pt := ADR(oct);
stop := LEN(oct);
FOR I := 1 TO stop DO
	(* read the first character and subtract 48 to get value in decimal 0 = 48 *)
	x := pt^;
	(* calculate the value of the digit *)
	IF X > 47 AND x < 56 THEN
		OCT_TO_BYTE := SHL(OCT_TO_BYTE,3) + X - 48;
	END_IF;
	pt := pt + 1;
END_FOR;



(* revision histroy
hm	18. jun. 2008	rev 1.0
	original release

hm	20. sep. 2008	rev 1.1
	changed length of input string from 20 to 10

*)

END_FUNCTION

// POUs/String/HEX_TO_BYTE
FUNCTION HEX_TO_BYTE : BYTE
VAR_INPUT
	HEX : STRING(5);
END_VAR
VAR
	pt : POINTER TO BYTE;
	i: INT;
	X: BYTE;
	stop: INT;
END_VAR

(*
version 1.1	20. sep. 2008
programmer 	hugo
tested by		oscat

HEX_TO_BYTE converts a Hexadecimal string into a byte.

*)

pt := ADR(hex);
stop := LEN(hex);
FOR I := 1 TO stop DO
	(* read the first character and subtract 48 to get value in decimal 0 = 48 *)
	x := pt^;
	(* calculate the value of the digit *)
	IF X > 47 AND x < 58 THEN
		HEX_TO_BYTE := SHL(HEX_TO_BYTE,4) + X - 48;
	ELSIF X > 64 AND X < 71 THEN
		HEX_TO_BYTE := SHL(HEX_TO_BYTE,4) + X - 55;
	ELSIF X > 96 AND X < 103 THEN
		HEX_TO_BYTE := SHL(HEX_TO_BYTE,4) + X - 87;
	END_IF;
	pt := pt + 1;
END_FOR;




(* revision histroy
hm	18. jun. 2008	rev 1.0
	original release

hm	20. sep.2008	rev 1.1
	changed length of input string from 20 to 5

*)

END_FUNCTION

// POUs/String/FSTRING_TO_DT
FUNCTION FSTRING_TO_DT : DT
VAR_INPUT
	SDT : STRING(60);
	FMT : STRING(60);
END_VAR
VAR CONSTANT
	ignore: STRING(1) := '*';  (* ignore character is * *)
	fchar : STRING(1) := '#';  (* format character is # *)
END_VAR
VAR
	c: STRING(1);
	tmp: STRING(20);
	end: INT;
	dy : INT := 1970;
	dm : INT := 1;
	dd : INT := 1;
	th : INT;
	tm : INT;
	ts : INT;
END_VAR


(*
version 1.0	24. sep. 2008
programmer 	hugo
tested by	oscat

FSTRING_TO_DT converts Formatted String into a DT value.

*)

(* scan input string *)
WHILE fmt <> '' DO
	c := LEFT(fmt,1);
	IF c = ignore THEN
		(* skip ignore characters *)
		fmt := DELETE(fmt,1,1);
		sdt := DELETE(sdt,1,1);
	ELSIF C = fchar THEN
		(* format chracter found skip format char and read identifier *)
		(* store format identifier in c and skip to next char in fmt *)
		c := MID(fmt,1,2);
		fmt := DELETE(fmt,2,1);
		(* extract the substring until the end of sdt or to next char of fmt *)
		IF fmt = '' THEN
			tmp := sdt;
		ELSE
			(* serach for end of substring *)
			end := FIND(sdt, LEFT(fmt,1))-1;
			tmp := LEFT(sdt, end);
			sdt := DELETE(sdt, end,1);
		END_IF;
		(* extract information from substring *)
		IF c = 'Y' THEN
			dy := STRING_TO_INT(tmp);
			IF dy < 100 THEN dy := dy + 2000; END_IF;
		ELSIF c = 'M' THEN
			dm := STRING_TO_INT(tmp);
		ELSIF c = 'N' THEN
			dm := FSTRING_TO_MONTH(tmp,0);
		ELSIF c = 'D' THEN
			dd := STRING_TO_INT(tmp);
		ELSIF c = 'h' THEN
			th := STRING_TO_INT(tmp);
		ELSIF c = 'm' THEN
			tm := STRING_TO_INT(tmp);
		ELSIF c = 's' THEN
			ts := STRING_TO_INT(tmp);
		END_IF;
	ELSIF c = LEFT(sdt,1) THEN
		(* skip matching characters *)
		fmt := DELETE(fmt,1,1);
		sdt := DELETE(sdt,1,1);
	ELSE
		RETURN;
	END_IF;
END_WHILE;

FSTRING_TO_DT := SET_DT(dy,dm,dd,th,tm,ts);


(* revision histroy
hm	24. sep. 2008	rev 1.0
	original release


*)

END_FUNCTION

// POUs/String/FSTRING_TO_MONTH
FUNCTION FSTRING_TO_MONTH : INT
VAR_INPUT
	MTH : STRING(20);
	LANG : INT;
END_VAR
VAR
	lx: INT;
END_VAR


(*
version 1.2	25. oct 2008
programmer 	hugo
tested by	oscat

FSTRING_TO_MONTH converts a string into a month, the string can be a name for the month or a number.
the function is language sensitve when LANG > 1 and checks for all languages when LANG = 0

*)

IF LANG = 0 THEN lx := LANGUAGE.DEFAULT; ELSE lx := MIN(LANG, LANGUAGE.LMAX); END_IF;
MTH := TRIM(mth);
MTH := CAPITALIZE(LOWERCASE(MTH));

FOR FSTRING_TO_MONTH := 1 TO 12 DO
	IF MTH = language.MONTHS[lx, FSTRING_TO_MONTH] THEN RETURN; END_IF;
	IF MTH = language.MONTHS3[lx, FSTRING_TO_MONTH] THEN RETURN; END_IF;
END_FOR;

(* since no name matched try to decode as integer *)
FSTRING_TO_MONTH := STRING_TO_INT(MTH);




(* revision histroy
hm	25. sep. 2008	rev 1.0
	original release

hm	19. oct. 2008	rev 1.1
	changed language setup constants

hm	25. oct. 2008	rev 1.2
	optimized code
*)

END_FUNCTION

// POUs/String/FSTRING_TO_DWORD
FUNCTION FSTRING_TO_DWORD : DWORD
VAR_INPUT
	IN : STRING(40);
END_VAR


(*
version 1.1	20. sep. 2008
programmer 	hugo
tested by		oscat

FSTRING_TO_BYTE converts a formatted string into a byte.
the string can be of the form 2#01010, 8#7234, 16#2AD3 and 1234

*)

IF LEFT(IN, 2) = '2#' THEN
	(* we need to convert binary *)
	FSTRING_TO_DWORD := BIN_TO_DWORD(RIGHT(in, LEN(in) - 2));
ELSIF LEFT(in, 2) = '8#' THEN
	(* weneed to convert octals *)
	FSTRING_TO_DWORD := OCT_TO_DWORD(RIGHT(in, LEN(in) - 2));
ELSIF LEFT(in, 3) = '16#' THEN
	(* we need to convert hexadecimal *)
	FSTRING_TO_DWORD := HEX_TO_DWORD(RIGHT(in, LEN(in) - 3));
ELSE
	(* we assume decimal representation *)
	FSTRING_TO_DWORD := DEC_TO_DWORD(CLEAN(in,'0123456789'));
END_IF;


(* revision histroy
hm	18. jun. 2008	rev 1.0
	original release

hm	20. sep. 2008	rev 1.1
	changed length of input dtring from 20 to 40


*)

END_FUNCTION

// POUs/String/OCT_TO_DWORD
FUNCTION OCT_TO_DWORD : DWORD
VAR_INPUT
	OCT : STRING(20);
END_VAR
VAR
	pt : POINTER TO BYTE;
	i: INT;
	X: BYTE;
	stop: INT;
END_VAR

(*
version 1.0	18. jun 2008
programmer 	hugo
tested by	oscat

OCT_TO_DWORD converts a octagonal string into a dword.

*)

pt := ADR(oct);
stop := LEN(oct);
FOR I := 1 TO stop DO
	(* read the first character and subtract 48 to get value in decimal 0 = 48 *)
	x := pt^;
	(* calculate the value of the digit *)
	IF X > 47 AND x < 56 THEN
		OCT_TO_DWORD := SHL(OCT_TO_DWORD,3) + X - 48;
	END_IF;
	pt := pt + 1;
END_FOR;




(* revision histroy
hm	18. jun. 2008	rev 1.0
	original release


*)

END_FUNCTION

// POUs/String/HEX_TO_DWORD
FUNCTION HEX_TO_DWORD : DWORD
VAR_INPUT
	Hex : STRING(20);
END_VAR
VAR
	pt : POINTER TO BYTE;
	i: INT;
	X: BYTE;
	stop: INT;
END_VAR

(*
version 1.4	18. jun. 2008
programmer 	hugo
tested by	tobias

HEX_TO_DWORD converts a Hexadecimal string into a DWORD.

*)

pt := ADR(hex);
stop := LEN(hex);
FOR I := 1 TO stop DO
	(* read the first character and subtract 48 to get value in decimal 0 = 48 *)
	x := pt^;
	(* calculate the value of the digit *)
	IF X > 47 AND x < 58 THEN
		HEX_TO_DWORD := SHL(HEX_TO_DWORD,4) + X - 48;
	ELSIF X > 64 AND X < 71 THEN
		HEX_TO_DWORD := SHL(HEX_TO_DWORD,4) + X - 55;
	ELSIF X > 96 AND X < 103 THEN
		HEX_TO_DWORD := SHL(HEX_TO_DWORD,4) + X - 87;
	END_IF;
	pt := pt + 1;
END_FOR;



(* revision histroy
hm	2.10.2007		rev 1.0
	original release

hm	19.11.2007		rev 1.1
	changed type of function from int to dword

hm 	4. mar 2008		rev 1.2
	added support for a..f and return 0 for invalid string

hm	29. mar. 2008	rev 1.3
	changed STRING to STRING(8)

hm	18. jun. 2008	rev 1.4
	changed input hex to STRING(20)
	function now ignores wrong characters
*)

END_FUNCTION

// POUs/String/FSTRING_TO_WEEK
FUNCTION FSTRING_TO_WEEK : BYTE
VAR_INPUT
	WEEK : STRING(60);
	LANG : INT;
END_VAR
VAR
	pos: INT;
END_VAR


(*
version 1.1	25. oct. 2008
programmer 	hugo
tested by	oscat

FSTRING_TO_WEEK converts a list of weekdays into a byte where each bit represents a day of the week.
bit 6 = mo, 0 = su;

*)

pos := FIND(WEEK, ',');
WHILE pos > 0 DO
	FSTRING_TO_WEEK := FSTRING_TO_WEEK OR SHR(BYTE#128, FSTRING_TO_WEEKDAY(MID(WEEK, pos - 1, 1), LANG));
	WEEK := RIGHT(WEEK, LEN(Week) - pos);
	pos := FIND(WEEK, ',');
END_WHILE;
FSTRING_TO_WEEK := (FSTRING_TO_WEEK OR SHR(BYTE#128, FSTRING_TO_WEEKDAY(WEEK, LANG))) AND BYTE#127;


(* revision histroy
hm	18. jun. 2008	rev 1.0
	original release

hm	25. oct. 2008	rev 1.1
	using language defauls and input lang
*)

END_FUNCTION

// POUs/String/FSTRING_TO_WEEKDAY
FUNCTION FSTRING_TO_WEEKDAY : INT
VAR_INPUT
	WDAY : STRING(20);
	LANG : INT;
END_VAR
VAR
	tmp: STRING(2);
	i: INT;
	ly: INT;
END_VAR


(*
version 1.2	25. oct. 2008
programmer 	hugo
tested by	oscat

FSTRING_TO_WEEKDAY converts a weekday string into an integer 1..7.

*)

IF LANG = 0 THEN ly := LANGUAGE.DEFAULT; ELSE ly := MIN(LANG, LANGUAGE.LMAX); END_IF;
(* tmp needs to be calculated first otherwise find can return wrong values *)
tmp := TRIM(wday);
tmp := CAPITALIZE(LOWERCASE(tmp));
FOR i := 1 TO 7 DO
	IF language.WEEKDAYS2[ly, i] = tmp THEN
		FSTRING_TO_WEEKDAY := i;
		RETURN;
	END_IF;
END_FOR;
FSTRING_TO_WEEKDAY := STRING_TO_INT(WDAY);




(* revision histroy
hm	18. jun. 2008	rev 1.0
	original release

hm	18. jul. 2008	rev 1.1
	changed nested call of left(trim()) for compatibility reasons

hm	25. oct. 2008	rev 1.2
	using language constants
*)

END_FUNCTION

// POUs/Mathematical/functions/FT_AVG
FUNCTION_BLOCK FT_AVG
VAR_INPUT
	IN : REAL;
	E : BOOL := TRUE;
	N : INT := 32;
	RST : BOOL;
END_VAR
VAR_OUTPUT
	AVG : REAL;
END_VAR
VAR
	buff : DELAY;
	i: INT;
	init : BOOL;
END_VAR

(*
version 1.5	10. mar. 2009
programmer 	hugo
tested by		oscat

this function calculates the moving average over n samples from a sequential input
the input values are shifted into an N deep buffer and the avg of this buffer is diplayed at anytime on the output.
a rst will load the buffer with the current in value..

*)

(* limit n to a max of 32 because delay can do max 32 cycles *)
buff.N := LIMIT(0, N, 32);

IF NOT init OR rst THEN
	FOR i := 1 TO N DO
		buff(in := in);
	END_FOR;
	avg := in;
	init := TRUE;
ELSIF E THEN
	buff(in := in);
	avg := avg + (in - buff.out ) / INT_TO_REAL(N);
END_IF;

(* revision history

hm	7. jan. 2007	rev 1.1
	chaged rst logic to load the buffer with the actual input value instead of 0.
	added en input to allow better control of signal flow
	added init to load the buffer with in at startup to avoid rampup at beginning.
	deleted unused variable cnt.

hm	14. jun. 2008	rev 1.2
	set default for input en = TRUE and N = 32

hm	10. oct. 2008	rev 1.3
	improved performance

hm	18. oct. 2008	rev 1.4
	changed input en to e for compatibility reasons

hm	10. mar. 2009	rev 1.5
	added type conversion for compatibility reasons

*)

END_FUNCTION_BLOCK

// POUs/Engineering/control/FT_IMP
FUNCTION_BLOCK FT_IMP
VAR_INPUT
	in : REAL;
	T : TIME;
	K : REAL := 1.0;
END_VAR
VAR_OUTPUT
	out : REAL;
END_VAR
VAR
	t1 : FT_PT1;
END_VAR

(*
version 1.1	3 Jan 2007
programmer 	hugo
tested by	oscat

FT_IMP is 	an impulse filter (high pass filter) with the time T and factor K.
 
*)

T1(in:= in, T:=T);
out := (in - t1.out) * K;

(*
hm 3.1.2007	rev 1.1
	added factor K

*)

END_FUNCTION_BLOCK

// POUs/Engineering/control/FT_INT2
FUNCTION_BLOCK FT_INT2
VAR_INPUT
	IN : REAL;
	K : REAL := 1.0;
	RUN : BOOL := TRUE;
	RST : BOOL;
	OUT_MIN : REAL := -1.0E38;
	OUT_MAX : REAL := 1.0E38;
END_VAR
VAR_OUTPUT
	OUT : REAL;
	LIM : BOOL;
END_VAR
VAR
	integ: INTEGRATE;
	ix : REAL;
	val : REAL2;
END_VAR


(*
version 1.2	11. mar. 2009
programmer 	hugo
tested by		oscat

FT_int2 is an integrator with input IN and factor K.
integration is only done while run = true, if run is false integration is stopped and the out remains at the last value.
if run is left unconnected, run is considered true by the function block.
the out_min and out_max values can be set to ,imit the output value range. 
the default for K is 1.
FT_INT2 has double presision accuracy (14 digits).


*)

IF RST THEN
	val := R2_SET(0.0);
	out := 0.0;
ELSE
	integ(X := IN, E := RUN, K := K, Y := ix);
	val := R2_ADD(val, ix);
	ix := 0.0;
	OUT := val.RX;
END_IF;

(* check output for limits *)
IF out > OUT_MIN AND out < OUT_MAX THEN
	LIM := FALSE;
ELSE
	OUT := LIMIT(OUT_MIN, OUT, OUT_MAX);
	val := R2_SET(OUT);
	LIM := TRUE;
END_IF;



(*	revision history
hm	2. jun. 2008	rev 1.0
	original version

hm	5. nov. 2008	rev 1.1
	rewritten code using integrate

hm	11. mar. 2009	rev 1.2
	real constants updated to new systax using dot

*)

END_FUNCTION_BLOCK

// POUs/Mathematical/Double Precision/R2_SET
FUNCTION R2_SET : REAL2
VAR_INPUT
	X : REAL;
END_VAR


(*
version 1.1	10. mar. 2009
programmer 	hugo
tested by		tobias

R2_set sets a double precision real to a single real value.

*)

R2_SET.RX := X;
R2_SET.R1 := 0.0;


(* revision history
hm	2. jun. 2008	rev 1.0
	original version

hm	10. mar. 2009	rev 1.1
	real constants updated to new systax using dot

*)

END_FUNCTION

// POUs/Mathematical/functions/FT_MIN_MAX
FUNCTION_BLOCK FT_MIN_MAX
VAR_INPUT
	in : REAL;
	rst : BOOL;
END_VAR
VAR_OUTPUT
	mx : REAL;
	mn : REAL;
END_VAR
VAR
	init: BOOL;
END_VAR

(*
version 1.0	1 sep 2006
programmer 	hugo
tested by		tobias

this function block stores the min and max value of an input signal.
when rst is true the mn and mx outputs are set to the in value.
when a rst is never active the function autoresets to the in value at startup.
since the input might not be present at first cycle the mn and mx are set during second cycle.

*)

IF rst OR NOT init THEN
	mn := in;
	mx := in;
	init := TRUE;
ELSIF in < mn THEN mn := in;
ELSIF in > mx THEN mx := in;
END_IF;

END_FUNCTION_BLOCK

// POUs/Engineering/control/FT_PD
FUNCTION_BLOCK FT_PD
VAR_INPUT
	IN : REAL;
	KP : REAL := 1.0;
	TV : REAL := 1.0;
END_VAR
VAR_OUTPUT
	Y : REAL;
END_VAR
VAR
	diff : FT_DERIV;
END_VAR

(*
version 1.0	3. jun 2008
programmer 	hugo
tested by		tobias

FT_PD is a PD controller.
The PD controller works according to the fomula Y = KP *(IN + DERIV(e) ).

*)

(* run differentiator *)
diff(IN := IN, K := TV);

(* combine both values *)
Y := KP * (diff.out + IN);



(* revision history
hm 	3. jun. 2008 	rev 1.0
	original version


*)

END_FUNCTION_BLOCK

// POUs/Engineering/control/FT_PDT1
FUNCTION_BLOCK FT_PDT1
VAR_INPUT
	IN : REAL;
	KP : REAL := 1.0;
	TV : REAL := 1.0;
	T1 : REAL := 1.0;
END_VAR
VAR_OUTPUT
	Y : REAL;
END_VAR
VAR
	diff : FT_DERIV;
	TP : FT_PT1;
END_VAR

(*
version 1.0	3. jun 2008
programmer 	hugo
tested by		tobias

FT_PD is a PD controller.
The PD controller works according to the fomula Y = KP *(IN + DERIV(e) ).

*)

(* run differentiator *)
diff(IN := IN, K := TV);

(* Run PT1 filter *)
tp(in := diff.out, T := REAL_TO_TIME(T1));

(* combine both values *)
Y := KP * (tp.out + IN);



(* revision history
hm 	3. jun. 2008 	rev 1.0
	original version


*)

END_FUNCTION_BLOCK

// POUs/Engineering/control/FT_PID
FUNCTION_BLOCK FT_PID
VAR_INPUT
	IN : REAL;
	KP : REAL := 1.0;
	TN : REAL := 1.0;
	TV : REAL := 1.0;
	ILIM_L : REAL := -1.0E38;
	ILIM_H : REAL := 1.0E38;
	IEN : BOOL := TRUE;
	RST : BOOL;
END_VAR
VAR_OUTPUT
	Y : REAL;
	LIM : BOOL;
END_VAR
VAR
	integ : FT_INT;
	diff : FT_DERIV;
END_VAR

(*
version 2.1	11. mar. 2009
programmer 	hugo
tested by		tobias

FT_PI is a PI controller.
The PID controller works according to the fomula Y = IN *(KP+ KI * INTEG(e) ).
a rst will reset the integrator to 0
ilim_h and iLim_l set the possible output range of the internal integrator.
the output flags lim will signal that the output limits are active.

default values for KP = 1, KI = 1, ILIM_L = -1E37, iLIM_H = +1E38.
*)

(* run integrator only if TN > 0 *)
IF TN > 0.0 THEN
	integ(IN := IN, K := 1.0 / TN, RUN := IEN, RST := RST, OUT_MIN := ILIM_L, OUT_MAX := ILIM_H);
ELSE
	integ(RST := FALSE);
END_IF;

(* run differentiator *)
diff(IN := IN, K := TV);

(* combine both values *)
Y := KP * (integ.Out + diff.out + IN);

(* check if integrator has reached its limits and set overflow *)
LIM := integ.LIM;



(* revision history
hm 3. jun. 2008 	rev 2.0
	original version

hm	11. mar. 2009	rev 2.1
	real constants updated to new systax using dot

*)

END_FUNCTION_BLOCK

// POUs/Engineering/control/FT_PIDW
FUNCTION_BLOCK FT_PIDW
VAR_INPUT
	IN : REAL;
	KP : REAL := 1.0;
	TN : REAL := 1.0;
	TV : REAL := 1.0;
	LIM_L : REAL := -1.0E38;
	LIM_H : REAL := 1.0E38;
	RST : BOOL;
END_VAR
VAR_OUTPUT
	Y : REAL;
	LIM : BOOL;
END_VAR
VAR
	integ : INTEGRATE;
	diff : FT_DERIV;
	YI: REAL;
END_VAR

(*
version 1.2	11. mar. 2009
programmer 	hugo
tested by		oscat

FT_PIDW is a PID controller with dynamic wind_up reset.
The PID controller works according to the fomula Y = KP *(IN + KI * INTEG(e) + DERIV(e) ).
a rst will reset the integrator to 0
lim_h and Lim_l set the possible output range of the internal integrator.
the output flags lim will signal that the output limits are active.

default values for KP = 1, KI = 1, ILIM_L = -1E37, iLIM_H = +1E38.
*)

(* run the integrator *)
IF tn = 0.0 OR rst THEN
	integ(E := FALSE, Y := YI);
	YI := 0.0;
ELSE
	integ(X := IN, K := 1.0 / TN, E := NOT LIM, Y := YI);
END_IF;

(* add up integrator and linear part *)
Y := KP * (IN + YI);

(* run differentiator *)
diff(IN := IN, K := TV);

(* set lim before differentiator is added to stop integrator if necessary *)
IF Y > LIM_L AND Y < LIM_H THEN
	LIM := FALSE;
ELSE
	LIM := TRUE;
END_IF;

(* add differential part and limit output Y *)

Y := LIMIT(LIM_L, Y + KP * diff.out, LIM_H);




(* revision history
hm 3. jun. 2008 	rev 1.0
	original version

hm	5. nov. 2008	rev 1.1
	changed code to use integrate

hm	11. mar. 2009	rev 1.2
	real constants updated to new systax using dot

*)

END_FUNCTION_BLOCK

// POUs/Engineering/control/FT_PIW
FUNCTION_BLOCK FT_PIW
VAR_INPUT
	IN : REAL;
	KP : REAL := 1.0;
	KI : REAL := 1.0;
	LIM_L : REAL := -1E38;
	LIM_H : REAL := 1E38;
	RST : BOOL;
END_VAR
VAR_OUTPUT
	Y : REAL;
	LIM : BOOL;
END_VAR
VAR
	integ : FT_INT;
END_VAR

(*
version 1.0	3. jun 2008
programmer 	hugo
tested by		tobias

FT_PIW is a PI controller.
The PID controller works according to the fomula Y = IN *(KP+ KI * INTEG(e) ).
a rst will reset the integrator to 0
ilim_h and iLim_l set the possible output range of the internal integrator.
the output flag lim will signal that the output limits are active.
the controller is equipped with anti wind_up circuitry that stops the integrator when lim_h or lim_l is reached


default values for KP = 1, KI = 1, ILIM_L = -1E37, iLIM_H = +1E38.
*)

(* run integrator *)
integ(IN := IN, K := KI, RUN := NOT LIM, RST := RST);

(* set output value *)
Y := KP * IN + integ.Out;

(* check for limits and set integrator for anti wind up *)
IF Y < LIM_L THEN
	Y := LIM_L;
	LIM := TRUE;
ELSIF Y > LIM_H THEN
	Y := LIM_H;
	LIM := TRUE;
ELSE
	LIM := FALSE;
END_IF;



(* revision history
hm 	3. jun. 2008 	rev 1.0
	original version


*)

END_FUNCTION_BLOCK

// POUs/Engineering/automation/FT_Profile
FUNCTION_BLOCK FT_Profile
VAR_INPUT
	K : REAL := 1.0;
	O : REAL;
	M : REAL := 1.0;
	E : BOOL;
END_VAR
VAR_INPUT CONSTANT
	value_0 : REAL;
	time_1 : TIME;
	value_1 : REAL;
	time_2 : TIME;
	value_2 : REAL;
	time_3 : TIME;
	value_3 : REAL;
	time_10 : TIME;
	value_10 : REAL;
	time_11 : TIME;
	value_11 : REAL;
	time_12 : TIME;
	value_12 : REAL;
	time_13 : TIME;
	value_13 : REAL;
END_VAR
VAR_OUTPUT
	Y : REAL;
	RUN : BOOL;
	ET : TIME;
END_VAR
VAR
	tx : TIME;
	edge : BOOL;
	state: BYTE;
	ta: TIME;
	tb: TIME;
	t0 : TIME;
	temp: REAL;
	va: REAL;
	vb: REAL;
END_VAR

(*
version 1.1	15 sep 2007
programmer 	tobias
tested by		hugo

FT_Profile generates an output signal which is defined by values over a time scale.
the different values are connected by ramps between the individual values.
a rising edge on E starts the output signal generation and E = True can delay time_3 / value_3 as long as it stays true.
an additional multiplier K can be used to multiply the output and an offset O can be added to the output dynamically.
*)

(* read system time *)
tx := DWORD_TO_TIME(T_PLC_MS());

(* determine start condition *)
IF E AND NOT edge THEN
	RUN := TRUE;
	ET := t#0s;
	t0 := tx;
	ta := tx;
	tb := multime(time_1, M);
	va := value_0;
	vb := value_1;
	temp := value_0;
	state := 1;
END_IF;
edge := E;

(* generate startup profile *)
IF run THEN
	CASE state OF
		1:	IF tx - ta >= tb THEN
				ta := ta + tb;
				tb := multime(time_2 - time_1, M);
				va := value_1;
				vb := value_2;
				temp := value_1;
				state := 2;
			ELSE
				temp := ((vb - va) * TIME_TO_REAL(tx - ta) / TIME_TO_REAL(tb) + va);
			END_IF;
		2:	IF tx - ta >= tb THEN
				ta := ta + tb;
				tb := multime(time_3 - time_2, M);
				va := value_2;
				vb := value_3;
				temp := value_2;
				state := 3;
			ELSE
				temp := ((vb - va) * TIME_TO_REAL(tx - ta) / TIME_TO_REAL(tb) + va);
			END_IF;
		3:	IF tx - ta >= tb THEN
				ta := ta + tb;
				tb := multime(time_10 - time_3, M);
				va := value_3;
				vb := value_10;
				temp := value_3;
				state := 4;
			ELSE
				temp := ((vb - va) * TIME_TO_REAL(tx - ta) / TIME_TO_REAL(tb) + va);
			END_IF;
		4 :	IF tx - ta >= tb THEN
				ta := ta + tb;
				tb := multime(time_11 - time_10, M);
				va := value_10;
				vb := value_11;
				temp := value_10;
				IF E THEN state := 5; ELSE state := 6; END_IF;
			ELSE
				temp := ((vb - va) * TIME_TO_REAL(tx - ta) / TIME_TO_REAL(tb) + va);
			END_IF;
		5:	(* extend the signal while E is true *)
			IF E THEN
				ta := tx;
			ELSE
				state := 6;
			END_IF;
		6:	IF tx - ta >= tb THEN
				ta := ta + tb;
				tb := multime(time_12 - time_11, M);
				va := value_11;
				vb := value_12;
				temp := value_11;
				state := 7;
			ELSE
				temp := ((vb - va) * TIME_TO_REAL(tx - ta) / TIME_TO_REAL(tb) + va);
			END_IF;
		7:	IF tx - ta >= tb THEN
				ta := ta + tb;
				tb := multime(time_13 - time_12, M);
				va := value_12;
				vb := value_13;
				temp := value_12;
				state := 8;
			ELSE
				temp := ((vb - va) * TIME_TO_REAL(tx - ta) / TIME_TO_REAL(tb) + va);
			END_IF;
		8:	IF tx - ta >= tb THEN
				temp := value_13;
				run := FALSE;
			ELSE
				temp := ((vb - va) * TIME_TO_REAL(tx - ta) / TIME_TO_REAL(tb) + va);
			END_IF;
	END_CASE;
	Y := temp * K + O;
	ET := tx - t0;
END_IF;

(* revision history
hm	27 feb 2007		rev 1.0
	original version

hm	15. sep2007		rev 1.1
	replaced Time() with T_PLC_MS for compatibility and performance reasons

*)

END_FUNCTION_BLOCK

// POUs/Engineering/control/FT_PT2
FUNCTION_BLOCK FT_PT2
VAR_INPUT
	in : REAL;
	T : TIME;
	D : REAL;
	K : REAL := 1.0;
END_VAR
VAR_OUTPUT
	out : REAL;
END_VAR
VAR
	init: BOOL;
	int1 : INTEGRATE;
	int2 : INTEGRATE;
	tn: REAL;
	I1, I2 : REAL;
	tn2: REAL;
END_VAR

(*
version 1.5	11. mar. 2009
programmer 	hugo
tested by		oscat

FT_PT2 is a 2nd grade filter with programmable times T, D and faktor K.
 
*)

(* startup initialisation *)
IF NOT init OR T = T#0s THEN
	init := TRUE;
	out := K * in;
	I2 := out;
ELSE
	TN := TIME_TO_REAL(T) * 1.0E-3;
	tn2 := TN * TN;
	int1(X := in * K / tn2 - I1 * 0.5 * D / TN - I2 / TN2, Y := I1);
	int2(X := I1,Y := I2);
	out := I2;
END_IF;


(* revision history

15.1.2007 hm		rev 1.1
	changed formula to new more acurate formula

hm 15.9.2007		rev 1.2
	deleted unused code for init system time reading tx	

hm	30.11.2007	rev 1.3
	changed out to be K * in during initialization
	avoind divide by 0 if tn = 0

hm	3. nov. 2008	rev 1.4
	optimized code and fixed a problem with init

hm	11. mar. 2009	rev 1.5
	real constants updated to new systax using dot

*)

END_FUNCTION_BLOCK

// POUs/Engineering/control/FT_TN16
FUNCTION_BLOCK FT_TN16
VAR_INPUT
	in : REAL;
	T : TIME;
END_VAR
VAR_OUTPUT
	out : REAL;
	trig : BOOL;
END_VAR
VAR
	length : INT := 16;
	X : ARRAY[0..15] OF REAL;
	cnt : INT;
	last : TIME;
	tx: TIME;
	init: BOOL;
END_VAR

(*
version 1.1	16 sep 2007
programmer 	hugo
tested by		tobias

FT_TN16 is delay function, it will delay a signal by a specified time : T and will store 16 values of in before they are put thru to out.
for higher or lower resolution please use FT_TN8 or FT_TN64 instead.
 
*)

(* read system time *)
tx := DWORD_TO_TIME(T_PLC_MS());

trig := FALSE;
IF NOT init THEN
	x[cnt] := in;
	init := TRUE;
	last := tx;
ELSIF tx - last >= T / length THEN
	IF cnt = length - 1 THEN cnt := 0; ELSE cnt := cnt + 1; END_IF;
	Out := X[cnt];
	x[cnt] := in;
	last := tx;
	Trig := TRUE;
END_IF;

(* revision history
hm		1. jan 2007	rev 1.0
	original version

hm		16. sep 2007	rev 1.1
	changes time() to T_plc_ms() for compatibility reasons

*)

END_FUNCTION_BLOCK

// POUs/Engineering/control/FT_TN8
FUNCTION_BLOCK FT_TN8
VAR_INPUT
	in : REAL;
	T : TIME;
END_VAR
VAR_OUTPUT
	out : REAL;
	trig: BOOL;
END_VAR
VAR
	length : INT := 8;
	X : ARRAY[0..7] OF REAL;
	cnt : INT;
	last : TIME;
	tx: TIME;
	init: BOOL;
END_VAR

(*
version 1.1	15 Sep 2007
programmer 	hugo
tested by		tobias

FT_TN8 is delay function, it will delay a signal by a specified time : T and will store 8 values of in before they are put thru to out.
if higher resolution is needed, pls use FT_TN16 or FT_TN64 instead.
 
*)

tx := DWORD_TO_TIME(T_PLC_MS());
trig := FALSE;
IF NOT init THEN
	x[cnt] := in;
	init := TRUE;
	last := tx;
ELSIF tx - last >= T / length THEN
	IF cnt = length - 1 THEN cnt := 0; ELSE cnt := cnt + 1; END_IF;
	Out := X[cnt];
	x[cnt] := in;
	last := tx;
	trig := TRUE;
END_IF;

(* revision history
hm		1. jan 2007		rev 1.0
	original version

hm		16. sep 2007	rev 1.1
	changes time() to T_plc_ms() for compatibility reasons

*)

END_FUNCTION_BLOCK

// POUs/Engineering/control/FT_TN64
FUNCTION_BLOCK FT_TN64
VAR_INPUT
	in : REAL;
	T : TIME;
END_VAR
VAR_OUTPUT
	out : REAL;
	trig: BOOL;
END_VAR
VAR
	length : INT := 64;
	X : ARRAY[0..63] OF REAL;
	cnt : INT;
	last : TIME;
	tx: TIME;
	init: BOOL;
END_VAR

(*
version 1.1	15 sep 2007
programmer 	hugo
tested by		tobias

FT_TN7 is delay function, it will delay a signal by a specified time : T and will store 64 values of in before they are put thru to out.
if lower resolution is needed, pls use FT_TN8 or FT_TN16 instead.
 
*)

(* read system time *)
tx := DWORD_TO_TIME(T_PLC_MS());

trig := FALSE;
IF NOT init THEN
	x[cnt] := in;
	init := TRUE;
	last := tx;
ELSIF tx - last >= T / length THEN
	IF cnt = length - 1 THEN cnt := 0; ELSE cnt := cnt + 1; END_IF;
	Out := X[cnt];
	x[cnt] := in;
	last := tx;
	trig := TRUE;
END_IF;

(* revision history
hm		1. jan 2007		rev 1.0
	original version

hm		16. sep 2007	rev 1.1
	changes time() to T_plc_ms() for compatibility reasons

*)

END_FUNCTION_BLOCK

// POUs/Mathematical/GAUSS
FUNCTION GAUSS : REAL
VAR_INPUT
	X : REAL;
	U : REAL;
	SI: REAL;
END_VAR
VAR
	temp: REAL;
	si_inv: REAL;
END_VAR


(*
version 1.2	10. mar. 2009
programmer 	hugo
tested by		tobias

this function calculates the gaussian density function

*)

temp := X - U;
si_inv := 1.0  / si;
GAUSS := EXP(Temp * Temp * si_inv * SI_inv * - 0.5) * 0.39894228 * si_inv;



(* revision hisdtory
hm	6. apr. 2008	rev 1.0
	original version

hm	27. oct. 2008	rev 1.1
	optimized performance	

hm	10. mar. 2009	rev 1.2
	real constants updated to new systax using dot

*)

END_FUNCTION

// POUs/Mathematical/GAUSSCD
FUNCTION GAUSSCD : REAL
VAR_INPUT
	X : REAL;
	U : REAL;
	SI: REAL;
END_VAR


(*
version 1.1	10. mar. 2009
programmer 	hugo
tested by		tobias

this function calculates the gaussian cumulative distribution function

*)

GAUSSCD := (ERF((X - U) / (SI * 1.414213562)) + 1.0) * 0.5;



(* revision hisdtory
hm	6. apr. 2008	rev 1.0
	original version

hm	10. mar. 2009	rev 1.1
	real constants updated to new systax using dot

*)

END_FUNCTION

// POUs/Mathematical/GDF
FUNCTION GDF : REAL
VAR_INPUT
	X : REAL;
END_VAR


(*
version 1.2	10. mar. 2009
programmer 	hugo
tested by		tobias

this function calculates the Gudermannian function.

*)

IF X = 0.0 THEN
	GDF := 0.0;
ELSIF X > 15.0 THEN
	GDF := math.PI05;
ELSIF X < -15.0 THEN
	GDF := -math.PI05;
ELSE
	GDF := ATAN(EXP(X)) * 2.0 - math.PI05;
END_IF;

(* revision history
hm	27. apr. 2008	rev 1.0
	original version

hm	18. oct. 2008	rev 1.1
	using math constants

hm	10. mar. 2009	rev 1.2
	real constants updated to new systax using dot

*)

END_FUNCTION

// POUs/Logic/generators/GEN_BIT
FUNCTION_BLOCK GEN_BIT
VAR_INPUT
	in0 : DWORD;
	in1 : DWORD;
	in2 : DWORD;
	in3 : DWORD;
	clk : BOOL;
	steps : INT;
	rep : INT;
	rst : BOOL;
END_VAR
VAR_OUTPUT
	Q0 :BOOL;
	Q1 :BOOL;
	Q2 :BOOL;
	Q3 :BOOL;
	cnt : INT;
	run : BOOL;
END_VAR
VAR
	r0: DWORD;
	r1: DWORD;
	r2: DWORD;
	r3: DWORD;
	rx : INT := 1;
END_VAR

(*
version 1.2	14. mar. 2009
programmer 	hugo
tested by		tobias

gen_bit is 4 bit sequencial pattern generator with 4 DWORD inputs and 4 serial outputs.
with the first clock pulse after a reset or after power on, bit 0 of the input DWORDS IN is present on the Outputs Q and the next clock cycle shifts to Bit 1 and so on.
the input steps defines how many bits of the input dwords will be shifted to the outputs. the sequence can be repetive when rep = 0 or any amount of repetitions can be defined with input rep.

*)

(* check if number of runs is finished or rep = 0 which means continuous *)

IF clk AND NOT rst THEN
	run := (rep = 0) OR (rx <= rep);
	IF run THEN
		(* check for step counter reached and reset to 0 if cnt = steps *)
		IF cnt = steps THEN
			cnt := 0;
		END_IF;

		(* when cnt = 0 then reload the inputs into the registers *)
		IF cnt = 0 THEN
			r0 := in0;
			r1 := in1;
			r2 := in2;
			r3 := in3;
		END_IF;

		(* when cnt < steps, shift the lowest bits to the outputs *)
		IF (cnt < steps) THEN
			Q0 := r0.0;
			Q1 := r1.0;
			Q2 := r2.0;
			Q3 := r3.0;
			r0 := SHR(r0,1);
			r1 := SHR(r1,1);
			r2 := SHR(r2,1);
			r3 := SHR(r3,1);
		END_IF;

		(* increment the step counter *)
		cnt := cnt +1;
		IF (cnt = steps) AND (rep <> 0) THEN rx := rx +1; END_IF;
		IF (rx > rep) AND (rep <> 0) THEN run := FALSE; END_IF;
	END_IF;
ELSE
	IF rst THEN
		run := FALSE;
		Q0 := FALSE;
		Q1 := FALSE;
		Q2 := FALSE;
		Q3 := FALSE;
		r0 := 0;
		r1 := 0;
		r2 := 0;
		r3 := 0;
		cnt := 0;
		rx := 1;
	END_IF;
END_IF;



(* revision histroy
hm	4 aug 2006	rev 1.0
	original version

hm 15. oct. 2008	rev 1.1
	improved performance

hm	14. mar. 2009	rev 1.2
	removed double assignments

*)

END_FUNCTION_BLOCK

// POUs/Engineering/signal generators/GEN_PW2
FUNCTION_BLOCK GEN_PW2
VAR_INPUT
	ENQ : BOOL;
	TH1 : TIME;
	TL1 : TIME;
	TH2 : TIME;
	TL2 : TIME;
	TS : BOOL;
END_VAR
VAR_OUTPUT
	Q : BOOL;
	TH : TIME;
	TL : TIME;
END_VAR
VAR
	t_high : TIME;
	t_low : TIME;
	tx : TIME;
	start : TIME;
	init : BOOL;
	et : TIME;
END_VAR

(*
version 1.1	14. mar. 2009
programmer 	hugo
tested by		oscat

GEN_PW2 generates a time TH? followed by a time TL?.
the input ts selects between 2 sets of timings for the operation.


*)

(* read system timer *)
tx := DWORD_TO_TIME(T_PLC_MS());

(* startup initialization *)
IF NOT init THEN
	start := tx;
	init := TRUE;
	TH := T#0s;
	TL := T#0s;
END_IF;

(* timing selection *)
IF TS THEN
	t_high := TH2;
	t_low := TL2;
ELSE
	t_high := TH1;
	t_low := TL1;
END_IF;

(* normal operation *)
IF ENQ THEN
	et := tx - start;
	IF NOT Q THEN
		IF et >= t_low THEN
			Q := TRUE;
			start := tx;
			TL := T#0s;
		ELSE
			TL := et;
		END_IF;
	ELSE
		IF et >= t_high THEN
			Q := FALSE;
			start := tx;
			TH := T#0s;
		ELSE
			TH := et;
		END_IF;
	END_IF;
ELSE
	Q := FALSE;
	TH := T#0s;
	TL := T#0s;
	start := tx;
END_IF;



(* revision history
hm	26. sep. 2008	rev 1.0
	original version

hm	14. mar. 2009	rev 1.1
	removed double assignments

*)

END_FUNCTION_BLOCK

// POUs/Engineering/signal generators/GEN_RDM
FUNCTION_BLOCK GEN_RDM
VAR_INPUT
	PT : TIME;
	AM : REAL := 1;
	OS : REAL;
END_VAR
VAR_OUTPUT
	Q : BOOL;
	Out : REAL;
END_VAR
VAR
	tx : TIME;
	last : TIME;
	init : BOOL;
END_VAR

(*
	version 1.1	16 sep 2007
	programmer 	oscat
	tested BY		oscat

this signal generator generates a random output. The signal is defined by period time (PT), 
amplitude (AM), offset (OS).
The Output waveform will have its max peak at AM/2 + OS and its minimum peak at -AM/2 + OS. 
The period time PT defines how often the output signal will jump to a new randow value.
The Output Q will be true for one cycle anytime the output OUT has changed

*)

(* read system time and prepare input data *)
tx := DWORD_TO_TIME(T_PLC_MS()) - last;

(* init section *)
IF NOT init THEN
	init := TRUE;
	last := tx;
	tx := t#0s;
END_IF;

(* add last if one cycle is finished *)
IF tx >= pt THEN
	last := last + pt;
	tx := tx - pt;

	(* generate output signal *)
	out := am * (RDM(0) - 0.5) + os;
	q := TRUE;
ELSE
	q := FALSE;
END_IF;

(* revision history

hm	7.2.2007		rev 1.0
	original version

hm	16.9.2007		rev 1.1
	changes time() to T_plc_ms() for compatibility reasons

*)

END_FUNCTION_BLOCK

// POUs/Engineering/signal generators/GEN_RDT
FUNCTION_BLOCK GEN_RDT

VAR_INPUT
	Enable		 : BOOL := TRUE ;
	Min_Time_ms	: TIME := t#1s ; (* min Taktzeit *)
	Max_Time_ms	: TIME := t#1.2s ; (* Max Taktzeit *)
	TP_Q		 : TIME := t#100ms ; (* Zeit Ausgang auf TRUE *)
END_VAR
VAR_OUTPUT
	xQ		 : BOOL ;
END_VAR
VAR
	(* Taktgenerator Simulation *)
	tonRDMTimer	: TON ; (* Zeitbaustein Taktgenerator *)
	tof_xQ		: TOF ; (* Ausschaltverzögerung Taktgenerator *)
	tRDMTime	: TIME ; (* Sollzeit *)
	rRDMTime	: REAL ; (* Zufalswert Timer *)
END_VAR

(*
version 1.1	16 mar. 2008
programmer 	J. Schohaus
tested by		Hugo

RDMT generates a defined pulse with pulse width TP_Q at random times. the random time will be defined with an minimum and maximum time.

*)


(*
FUNCTION_BLOCK RDMTimer
###############################################################################
		 Ersteller / author :		 		 		 		 		 J.Schohaus
		 Datum / date:		 		 		 		 		 		 13.07.2007
###############################################################################
		 Änderungen / Datum / Ersteller :		 		 		 		 		 		 		 		 		 		 		 		 		 		 		 
		 moditication / date / author :		 		 
###############################################################################
		 Verwendete Bibliotheken		 ( * werden im Baustein nicht benötigt )
		 		 		 		 Oscat.lib
###############################################################################
Beschreibung:
*)

tonRDMTimer ( IN:= Enable , PT:= tRDMTime );
tof_xQ ( IN:= tonRDMTimer.Q , PT:= TP_Q );
XQ := tof_xq.Q;
IF tonRDMTimer.Q THEN
		 xQ := TRUE ;
		 rRDMTime := RDM ( last:= rRDMTime ) ;
		 tRDMTime := REAL_TO_TIME ( rRDMTime * DINT_TO_REAL(TIME_TO_DINT( Max_Time_ms - Min_Time_ms ) + TIME_TO_DINT(Min_Time_ms ))) ;
		 tonRDMTimer ( IN:= FALSE );
END_IF;

(* revision history
J. Schohaus	19. nov 2007	rev 1.0
	origial version

hm	16. mar. 2008			rev 1.1
	added type conversion to avoid warnings under codesys 3.0
*)

END_FUNCTION_BLOCK

// POUs/Engineering/signal generators/GEN_RMP
FUNCTION_BLOCK GEN_RMP
VAR_INPUT
	PT : TIME := t#1s;
	AM : REAL := 1.0;
	OS : REAL;
	DL : REAL;
END_VAR
VAR_OUTPUT
	Q : BOOL;
	OUT : REAL;
END_VAR
VAR
	tx : TIME;
	last : TIME;
	init : BOOL;
	temp : REAL;
	ltemp: REAL;
END_VAR

(*
	version 1.4	10. mar. 2009
	programmer 	oscat
	tested BY		oscat

this signal generator generates a ramp wave output. The ramp wave signal is defined by period time (PT), 
amplitude (AM), offset (OS) and a specific delay for the output signal (DL).
The Output waveform will have its minimum peak at OS and its maximum peak at AM + OS. 
The delay input can delay a signal up to PT, this can be useful to synchronize different generators 
and generate interleaving signals.
in addition to the analog output Out there is a second boolean output Q with is true for one cycle when the ramp starts.
*)

(* read system time and prepare input data *)
tx := DWORD_TO_TIME(T_PLC_MS()) - last;
DL := MODR(dl,1.0);
IF dl < 0.0 THEN dl := 1.0 - dl; END_IF;

(* init section *)
IF NOT init THEN
	init := TRUE;
	last := tx;
	tx := t#0s;
END_IF;

(* add last if one cycle is finished *)
IF tx >= pt THEN
	last := last + pt;
	tx := tx - pt;
END_IF;

(* generate sine wave *)
ltemp := temp;
IF pt > t#0s THEN temp := FRACT(TIME_TO_REAL(tx + MULTIME(pt, dl)) / TIME_TO_REAL(pt)); END_IF;
out := am * temp + os;

(* boolean output Q *)
Q := temp < ltemp;

(* revision history
hm	3. mar 2007		rev 1.0
	original version

hm	17 sep 2007		rev 1.1
	replaced time() with t_plc_ms for compatibilitx reasons

hm	27. nov 2007	rev 1.2
	avoid divide by 0 when pt = 0

ks	26. oct. 2008	rev 1.3
	code optimization

hm	10. mar. 2009	rev 1.4
	changed real constants to use dot syntax
*)

END_FUNCTION_BLOCK

// POUs/Engineering/signal generators/GEN_SIN
FUNCTION_BLOCK GEN_SIN
VAR_INPUT
	PT : TIME;
	AM : REAL := 1.0;
	OS : REAL;
	DL : REAL;
END_VAR
VAR_OUTPUT
	Q : BOOL;
	Out : REAL;
END_VAR
VAR
	tx : TIME;
	last : TIME;
	init : BOOL;
	temp : REAL;
END_VAR

(*
version 1.6	11. mar. 2009
programmer 	oscat
tested BY	oscat

this signal generator generates a sine wave output. The sine wave signal is defined by period time (PT), 
amplitude (AM), offset (OS) and a specific delay for the output signal (DL).
The Output waveform will have its max peak at AM/2 + OS and its minimum peak at -AM/2 + OS. 
The delay input can delay a signal up to PT, this can be useful to synchronize different generators 
and generate interleaving signals. A Cos wave can be generated accordingly.
in addition to a analog output Out there is a second boolean output Q with the corresponding binary signal.
*)

(* read system time and prepare input data *)
tx := DWORD_TO_TIME(T_PLC_MS()) - last;
DL := MODR(dl,1.0);
IF dl < 0.0 THEN dl := 1.0 - dl; END_IF;

(* init section *)
IF NOT init THEN
	init := TRUE;
	last := tx;
	tx := t#0s;
END_IF;

(* add last if one cycle is finished *)
IF tx >= pt THEN
	last := last + pt;
	tx := tx - pt;
END_IF;

(* generate sine wave *)
IF pt > t#0s THEN temp := SIN(math.PI2 * DWORD_TO_REAL(TIME_TO_DWORD(tx + MULTIME(pt, dl))) / DWORD_TO_REAL(TIME_TO_DWORD(pt))); END_IF;
out := am * 0.5 *  temp + os;

(* boolean output Q *)
q := NOT SIGN_R(temp);

(* revision history
hm	22. jan 2007	rev 1.0
	original version

hm	17 sep 2007	rev 1.1
	replaced time() with t_plc_ms for compatibilitx reasons

hm	27. nov 2007	rev 1.2
	avoid divide by 0 when pt = 0

hm	6. jan 2008		rev 1.3
	improved performance

hm	16. mar. 2008	rev 1.4
	added type conversion to avoid warnings under codesys 3.0

hm	18. oct. 2008	rev 1.5
	using math constants

hm	11. mar. 2009	rev 1.6
	changed real constants to use dot syntax

*)

END_FUNCTION_BLOCK

// POUs/Logic/generators/GEN_SQ
FUNCTION_BLOCK GEN_SQ
VAR_INPUT
	PT : TIME;
END_VAR
VAR_OUTPUT
	Q : BOOL;
END_VAR
VAR
	tn: TIME;
	tx: TIME;
	init : BOOL;
END_VAR

(*
version 1.2	18. jul. 2009
programmer 	hugo
tested by		tobias

gen_sq generates square wave signal with programmable period time.

*)

(* read system time *)
tx := DWORD_TO_TIME(T_PLC_MS());

IF tx >= tn THEN
	Q := NOT Q;
	IF init THEN
		tn := tn + DWORD_TO_TIME(SHR(TIME_TO_DWORD(PT),1));
	ELSE
		tn := tx;
		init := TRUE;
	END_IF;
END_IF;

(* revision history
hm	4. aug 2006	rev 1.0
	original version

hm	17. sep 2007	rev 1.1
	replaced time() with T_PLC_MS() for compatibility reasons

hm	18. jul. 2009	rev 1.2
	improved accuracy

*)

END_FUNCTION_BLOCK

// POUs/Engineering/signal generators/GEN_SQR
FUNCTION_BLOCK GEN_SQR
VAR_INPUT
	PT : TIME;
	AM : REAL := 1.0;
	OS : REAL;
	DC : REAL := 0.5;
	DL : REAL;
END_VAR
VAR_OUTPUT
	Q : BOOL;
	Out : REAL;
END_VAR
VAR
	tx : TIME;
	last : TIME;
	init: BOOL;
END_VAR

(*
version 1.4	11. mar. 2009
programmer 	oscat
tested BY		oscat

this signal generator generates a square wave output. The square wave signal is defined by period time (PT), 
amplitude (AM), offset (OS), duty cycle (DC) and a specific delay for the output signal (DL).
The Output waveform will switch between AM/2 + OS and -AM/2 + OS. The DC input specifies ther duty cycle, 
DC = 0 means output is low at all times and 1 means output is high at all times.
The delay input can delay a signal up to PT, this can be useful to synchronize different generators and generate interleaving signals.
in addition to a analog output Out there is a second boolean output Q.
*)

(* check dc = 1 or 0 *)
IF dc = 0.0 THEN
	out := -am * 0.5 + os;
	Q := FALSE;
	RETURN;
ELSIF dc = 1.0 THEN
	out := am * 0.5 + os;
	Q := TRUE;
	RETURN;
END_IF;

(* read system time and prepare input data *)
tx := DWORD_TO_TIME(T_PLC_MS()) - last;
DL := MODR(dl,1.0);
IF dl < 0.0 THEN dl := 1.0 - dl; END_IF;
dc := MODR(dc,1.0);
IF dc < 0.0 THEN dc := 1.0 - dc; END_IF;

(* init section *)
IF NOT init THEN
	init := TRUE;
	last := tx;
	tx := t#0s;
END_IF;

(* add last if one cycle is finished *)
IF tx >= pt THEN
	last := last + pt;
	tx := tx - pt;
END_IF;

(* check if falling or rising edge first *)
IF MULTIME(pt, dl + dc) >= pt THEN
	(* generate falling edge *)
	IF tx >= MULTIME(pt, dl + dc - 1) THEN
		out := -am * 0.5 + os;
		Q := FALSE;
	END_IF;
	(* generate rising edge *)
	IF tx >= MULTIME(pt, dl) THEN
		out := am * 0.5 + os;
		Q := TRUE;
	END_IF;
ELSE
	(* generate rising edge first *)
	IF tx >= MULTIME(pt, dl) THEN
		out := am * 0.5 + os;
		Q := TRUE;
	END_IF;
	(* generate falling edge *)
	IF tx >= MULTIME(pt, dl + dc) THEN
		out := -am * 0.5 +os;
		Q := FALSE;
	END_IF;
END_IF;

(* revision history

hm	12. feb 2007	rev 1.1
	added default value for dc = 0.5

hm	17 sep 2007	rev 1.2
	replaced time() with t_plc_ms for compatibilitx reasons

hm	6. jan 2008	rev 1.3
	improved performance

hm	11. mar. 2009	rev 1.4
	changed real constants to use dot syntax
	set default amplitude to 1.0

*)

END_FUNCTION_BLOCK

// POUs/Engineering/conversion/GEO_TO_DEG
FUNCTION GEO_TO_DEG : REAL
VAR_INPUT
	D : INT;
	M : INT;
	SEC : REAL;
END_VAR


(*
version 1.0	22. jan. 2009
programmer 	hugo
tested by		oscat

this function converts degrees, minutes seconds to decimal degrees.

*)

GEO_TO_DEG := INT_TO_REAL(D) + INT_TO_REAL(M) * 0.016666666666667 + sec * 0.00027777777777778;


(* revision histroy
hm	22. jan. 2009	rev 1.0
	original release


*)

END_FUNCTION

// POUs/Mathematical/GOLD
FUNCTION GOLD : REAL
VAR_INPUT
	X : REAL;
END_VAR


(*
version 1.1	10. mar. 2009
programmer 	hugo
tested by		tobias

this function calculates the golden function.

*)

GOLD := (X + SQRT(X*X + 4.0)) * 0.5;


(* revision history
hm	27. apr. 2008	rev 1.0
	original version

hm	10. mar. 2009	rev 1.1
	real constants updated to new systax using dot

*)

END_FUNCTION

// POUs/Logic/gate logic/GRAY_TO_BYTE
FUNCTION GRAY_TO_BYTE : BYTE
VAR_INPUT
	IN : BYTE;
END_VAR


(*
version 1.0	9. nov. 2009
programmer 	hugo
tested by		oscat

this function converts a gray code into binary

*)

GRAY_TO_BYTE := SHR(IN,4) XOR IN;
GRAY_TO_BYTE := SHR(GRAY_TO_BYTE,2) XOR GRAY_TO_BYTE;
GRAY_TO_BYTE := SHR(GRAY_TO_BYTE,1) XOR GRAY_TO_BYTE;

(* revision history
hm	9. nov. 2009	rev 1.0
	original version

*)

END_FUNCTION

// POUs/Building/HLK/HEAT_INDEX
FUNCTION HEAT_INDEX : REAL
VAR_INPUT
	T : REAL;
	RH : REAL;
END_VAR
VAR
	RH2 : REAL;
	T2 : REAL;
END_VAR

(*
version 1.3	13. mar. 2009
programmer 	hugo
tested by		tobias

this function calculates the heat index temperature depending on external temperature and Relative humidity

*)

IF RH < 20.0 OR T < 20.0 THEN
	HEAT_INDEX := T;
ELSE
	RH2 := RH * RH;
	T := C_TO_F(T);
	T2 := T * T;
	HEAT_INDEX := -42.379 + 2.04901523 * T - 6.83783E-3 * T2
			+ RH * (10.1433127 - 0.22475541 * T + 1.22874E-3 * T2)
			+ RH2 * (8.5282E-4 * T - 5.481717E-2 - 1.99E-6 * T2);
	HEAT_INDEX := F_TO_C(HEAT_INDEX);
END_IF;

(* revision history

hm 27.2.2007		rev 1.1
	deleted unused variables rh3 and T3

hm	2.12.2007		rev 1.2
	changed code for better performance

hm	13. mar. 2009	rev 1.3
	real constants updated to new systax using dot

*)

END_FUNCTION

// POUs/Building/HLK/HEAT_METER
FUNCTION_BLOCK HEAT_METER
VAR_INPUT
	TF, TR : REAL;
	LPH : REAL;
	E : BOOL;
	RST : BOOL;
END_VAR
VAR_INPUT CONSTANT
	CP : REAL;
	Density : REAL;
	Content : REAL;
	Pulse_Mode : BOOL;
	Return_meter : BOOL;
	AVG_time : TIME := T#5s;
END_VAR
VAR_OUTPUT
	C : REAL;
END_VAR
VAR_IN_OUT
	Y : REAL;
END_VAR
VAR
	tx, last : DWORD;
	int1 : FT_INT2;
	edge : BOOL;
	x: REAL;
	init: BOOL;
	y_last: REAL;
END_VAR

(*
version 1.9	13. nov. 2009
programmer 	hugo
tested by		oscat

Heat meter measures the heat transfer of water of a mixture of water and another component.
The inputs are foreward temperature and reverse temperature.
the additional component is specified with its parameters density, Specific heat capacity and content in %.
an input e anables the measurement while it can be configured to be based on X liters / pulse or in liters / hour.
the output Y is in Joule.

*)

IF rst THEN
	int1(rst := TRUE);
	int1.rst := FALSE;
	C := 0.0;
	Y := 0.0;
ELSIF e THEN
	X := (WATER_DENSITY(SEL(return_meter, TF, TR), FALSE) * (WATER_ENTHALPY(TF) - WATER_ENTHALPY(TR)) * (1.0 - content) + CP * Density * content * (TF-TR));
END_IF;

(* integrate or add consumption *)
int1(run := NOT pulse_mode AND e, in := X * LPH * 2.77777777777E-4);
IF pulse_mode THEN
	IF NOT edge THEN Y := Y + X * LPH; END_IF;
ELSE
	Y := int1.Out;
END_IF;

(* store the value of e *)
edge := e;

(* read system_time *)
tx := T_PLC_MS();

(* only init at startup necessary *)
IF NOT init THEN
	init := TRUE;
	last := tx;
END_IF;

(* calculate the current consumption *)
IF (tx - last >= TIME_TO_DWORD(AVG_TIME)) AND (avg_time > T#0s) THEN
	last := tx;
	C := (Y - Y_last) * 3.6E6 / DWORD_TO_REAL(TIME_TO_DWORD(AVG_TIME));
	Y_last := Y;
END_IF;



(* revision history
hm	16. nov. 2007	rev 1.0
	original version

hm	24. dec. 2007	rev 1.1
	added config variable return_meter
	added output C for current consumption

hm	6. mar. 2008	rev 1.2
	corrected an error in pulse mode

hm	16. mar. 2008	rev 1.3
	added type conversion to avoid warnings under codesys 3.0

hm	21. oct. 2008	rev 1.4
	improved code

hm	6. nov. 2008	rev 1.5
	changed to FT_INT2 to avoid overrun at hig values

hm	8. feb. 2009	rev 1.6
	changes Y to be I/O

hm	23. mar. 2009	rev 1.7
	real constants updated to new systax using dot
	corected error in formula

hm	27. jul 2009	rev 1.8
	output C is now calculated in J/h

hm	13. nov. 2009	rev 1.9
	output C is now calculated correctly
*)

END_FUNCTION_BLOCK

// POUs/Building/HLK/WATER_DENSITY
FUNCTION WATER_DENSITY : REAL
VAR_INPUT
	T : REAL;
	Sat : BOOL;
END_VAR
VAR CONSTANT
	a0 : REAL := 999.83952;
	a1 : REAL := 16.952577;
	a2 : REAL := -7.9905127E-3;
	a3 : REAL := -4.6241757E-5;
	a4 : REAL := 1.0584601E-7;
	a5 : REAL := -2.8103006E-10;
	b  : REAL := 0.0168872;
END_VAR
VAR
	T2: REAL;
	T4: REAL;
END_VAR


(*
version 1.2	13. mar. 2009
programmer 	hugo
tested by		tobias

this function calculates the water density for air free water between 0 and 100 deg C
while sat is false the denisty is calculated for air free water and when sat = true
the calculation is performed for water saturated with air.

*)

T2 := T * T;
T4 := T2 * T2;
WATER_DENSITY := (a0 + a1*T + a2*T2 + a3*T2*T + a4*T4 + a5*T4*T) / (1.0 + b*T);
IF sat THEN WATER_DENSITY := WATER_DENSITY - 0.004612 + 0.000106 * T; END_IF;


(* revision history

hm	13.9.2007		rev 1.0
	original version

hm	2.12.2007		rev 1.1
	changed code for better performance

hm	13. mar. 2009	rev 1.2
	real constants updated to new systax using dot

*)

(*
    °C - die Celsius-Temperatur in Grad Celsius
    v  das spezifische Volumen in Kubikdezimeter je Kilogramm dm³/kg
    h  die spezifische Enthalpie in Kilojoule je Kilogramm 	kJ/kg
    u  die spezifische Innere Energie in Kilojoule je Kilogramm 	kJ/kg
    s  die spezifische Entropie in Kilojoule je Kilogramm mal Kelvin 	kJ/(kg·K)
    cp - die spezifische Wärmekapazität bei konstantem Druck in Kilojoule je Kilogramm mal Kelvin 	kJ/(kg·K)
    Y  Volumenausdehnungskoeffizient in 10-3 durch Kelvin  10-3/K
    L  Wärmeleitfähigkeit in Milliwatt je Meter mal Kelvin  mW / (m·K) 
    n  Viskosität in Mikropascal mal Sekunde uPa·s 	
    s ?  Oberflächenspannung in Millinewton je Meter  mN/m


°C 		v 				h 			u 		s 			cp 		Y 		L		n		s	
-20		1,006580	
0 		1,000160 		0,06 		-0,04 	-0,0001 	4,228 	-0,080 	561,0 	1792 	75,65
4		1,000028
5 		1,0000 		21,1 		21,0 	0,076 		4,200 	0,011 	570,6 	1518 	74,95
10 		1,0003 		42,1 		42,0 	0,151 		4,188 	0,087 	580,0 	1306 	74,22
15 		1,0009 		63,0 		62,9 	0,224 		4,184 	0,152 	589,4 	1137 	73,49
20 		1,001797 		83,9 		83,8 	0,296 		4,183 	0,209 	598,4 	1001 	72,74
25 		1,0029 		104,8 		104,7 	0,367 		4,183 	0,259 	607,2 	890,4 	71,98
30 		1,0044 		125,8 		125,7 	0,437 		4,183 	0,305 	615,5 	797,7 	71,20
35 		1,0060 		146,7 		146,6 	0,505 		4,183 	0,347 	623,3 	719,6 	70,41
40 		1,007842 		167,58 	167,5 	0,572 		4,182 	0,386 	630,6 	653,3 	69,60
45 		1,0099 		188,5 		188,4 	0,638 		4,182 	0,423 	637,3 	596,3 	68,78
50 		1,0121 		209,4 		209,3 	0,704 		4,181 	0,457 	643,6 	547,1 	67,95
60 		1,017089 		251,2 		251,1 	0,831 		4,183 	0,522 	654,4 	466,6 	66,24
70 		1,0227 		293,1 		293,0 	0,955 		4,187 	0,583 	663,1 	404,1 	64,49
80 		1,029027 		335,0 		334,9 	1,075 		4,194 	0,640 	670,0 	354,5 	62,68
90 		1,0359 		377,0 		376,9 	1,193 		4,204 	0,696 	675,3 	314,6 	60,82
99,63 	1,0431 		417,5 		417,4 	1,303 		4,217 	0,748 	679,0 	283,0 	58,99
100	1,043453		419,1

Stoffdaten von Wasser Quelle Wickipedia

*)

END_FUNCTION

// POUs/Building/HLK/WATER_ENTHALPY
FUNCTION WATER_ENTHALPY : REAL
VAR_INPUT
	T : REAL;
END_VAR
VAR
	Pts : INT := 11;
	data : ARRAY[1..20, 0..1] OF REAL :=[ 0.0,0.06, 10.0,42.1, 20.0,83.9, 30.0,125.8, 40.0,167.58, 50.0,209.4, 60.0,251.2, 70.0,293.1, 80.0,335.0, 90.0, 377.0, 100.0,419.1];
END_VAR

(*
version 1.1	13. mar. 2009
programmer 	hugo
tested by		tobias

water_enthalpy calculates the enthalpy of liquid water from 0..100 °C 

*)

WATER_ENTHALPY := LINEAR_INT(T, Data, Pts);



(*
    °C - die Celsius-Temperatur in Grad Celsius
    v  das spezifische Volumen in Kubikdezimeter je Kilogramm dm³/kg
    h  die spezifische Enthalpie in Kilojoule je Kilogramm 	kJ/kg
    u  die spezifische Innere Energie in Kilojoule je Kilogramm 	kJ/kg
    s  die spezifische Entropie in Kilojoule je Kilogramm mal Kelvin 	kJ/(kg·K)
    cp - die spezifische Wärmekapazität bei konstantem Druck in Kilojoule je Kilogramm mal Kelvin 	kJ/(kg·K)
    Y  Volumenausdehnungskoeffizient in 10-3 durch Kelvin  10-3/K
    L  Wärmeleitfähigkeit in Milliwatt je Meter mal Kelvin  mW / (m·K) 
    n  Viskosität in Mikropascal mal Sekunde uPa·s 	
    s ?  Oberflächenspannung in Millinewton je Meter  mN/m


°C 		v 				h 			u 		s 			cp 		Y 		L		n		s	
-20		1,006580	
0 		1,000160 		0,06 		-0,04 	-0,0001 	4,228 	-0,080 	561,0 	1792 	75,65
4		1,000028
5 		1,0000 		21,1 		21,0 	0,076 		4,200 	0,011 	570,6 	1518 	74,95
10 		1,0003 		42,1 		42,0 	0,151 		4,188 	0,087 	580,0 	1306 	74,22
15 		1,0009 		63,0 		62,9 	0,224 		4,184 	0,152 	589,4 	1137 	73,49
20 		1,001797 		83,9 		83,8 	0,296 		4,183 	0,209 	598,4 	1001 	72,74
25 		1,0029 		104,8 		104,7 	0,367 		4,183 	0,259 	607,2 	890,4 	71,98
30 		1,0044 		125,8 		125,7 	0,437 		4,183 	0,305 	615,5 	797,7 	71,20
35 		1,0060 		146,7 		146,6 	0,505 		4,183 	0,347 	623,3 	719,6 	70,41
40 		1,007842 		167,58 	167,5 	0,572 		4,182 	0,386 	630,6 	653,3 	69,60
45 		1,0099 		188,5 		188,4 	0,638 		4,182 	0,423 	637,3 	596,3 	68,78
50 		1,0121 		209,4 		209,3 	0,704 		4,181 	0,457 	643,6 	547,1 	67,95
60 		1,017089 		251,2 		251,1 	0,831 		4,183 	0,522 	654,4 	466,6 	66,24
70 		1,0227 		293,1 		293,0 	0,955 		4,187 	0,583 	663,1 	404,1 	64,49
80 		1,029027 		335,0 		334,9 	1,075 		4,194 	0,640 	670,0 	354,5 	62,68
90 		1,0359 		377,0 		376,9 	1,193 		4,204 	0,696 	675,3 	314,6 	60,82
99,63 	1,0431 		417,5 		417,4 	1,303 		4,217 	0,748 	679,0 	283,0 	58,99
100	1,043453		419,1

Stoffdaten von Wasser Quelle Wickipedia

Wasser hat unter Normaldruck seine größte Dichte von 1000 Kilogramm pro Kubikmeter bei 3,98 °C und zeigt damit eine Dichteanomalie. 
Diese besteht darin, dass sich Wasser unterhalb von 3,98 °C bei weiterer Temperaturverringerung, auch beim Wechsel zum festen 
Aggregatzustand, wieder ausdehnt, was man nur von wenigen Stoffen kennt. Die derzeit genauesten publizierten Werte für die maximale 
Dichte liegen bei (999,974950 ± 0,00084) kg/m³ und bei (3,983 ± 0,00067) °C für die Temperatur, bei der dieser Wert erreicht wird. 
Die Werte stellen einen Mittelwert der von verschiedenen physikalischen Instituten veröffentlichten Zahlen dar (Stand 2001).

Die Berechnung der Dichte von luftfreiem Wasser DLF in Abhängigkeit von der Temperatur T ([T] = °C) kann mit Hilfe der folgenden 
Virialgleichung erfolgen:
: \frac{D_{\rm LF}}{\rm g/l} = \frac{a_0 + a_1 T + a_2 T^2 + a_3 T^3 + a_4 T^4 + a_5 T^5}{1 + b T}.
mit den Koeffizienten: a0 = 999,83952; a1 = 16,952577 (°C)-1; a2 = -7,9905127·10-3 (°C)-2; a3 = -4,6241757·10-5 (°C)-3; 
a4 = 1,0584601·10-7 (°C)-4; a5 = -2,8103006·10-10 (°C)-5 und b = 0,0168872. 
Für die Berechnung der Dichte von luftgesättigtem Wasser korrigiert man den Wert nach 
DLG/(g/l) = DLF/(g/l) - 0,004612 + 0,000106 (°C)-1·T. (Quelle: PTB-Mitteilungen 100/3-90)

*)

(* revision history
hm	13. mar. 2009	rev 1.0
	original version

hm	13. mar. 2009	rev 1.1
	real constants updated to new systax using dot

*)

END_FUNCTION

// POUs/Mathematical/functions/LINEAR_INT
FUNCTION LINEAR_INT : REAL
VAR_INPUT
	X : REAL;
	XY : ARRAY[1..20,0..1] OF REAL;
	Pts : INT;
END_VAR
VAR
	i : INT;
END_VAR

(*
	version 1.1	27 dec 2007
	programmer 	oscat
	tested BY		oscat

LINEAR_INT calculates an output based on a linear interpolation of up to 20 coordinates given in an array
the input coordinates have to start at the lowest array position and must be sorted ba ascending X values.

*)

(*make sure n is bound within the array size *)
pts := MIN(pts,20);

(* calculate the linear segement interpolation *)
i := 2;
(* search for segment and calculate output
	below and above the defined segments we interpolate the last segment *)
WHILE (i < pts) AND (XY[i,0] < X) DO
	i := i + 1;
END_WHILE;

(* calculate the output value on the corresponding segment coordinates *)
LINEAR_INT := ((XY[i,1] - XY[i-1,1]) * X - XY[i,1] * XY[i-1,0] + XY[i-1,1] * XY[i,0]) / (XY[i,0] - XY[i-1,0]);

(* revision history
hm	7. oct 2007		rev 1.0
	original version

hm	27 dec 2007		rev 1.1
	changed code for better performance
*)

END_FUNCTION

// POUs/Building/HLK/HEAT_TEMP
FUNCTION_BLOCK HEAT_TEMP
VAR_INPUT
	T_EXT : REAL;
	T_INT : REAL;
	OFFSET : REAL;
	T_REQ : REAL;
END_VAR
VAR_INPUT CONSTANT
	TY_MAX : REAL := 70.0;
	TY_MIN : REAL := 25.0;
	TY_CONFIG : REAL := 70.0;
	T_INT_CONFIG : REAL := 20.0;
	T_EXT_CONFIG : REAL := -15.0;
	T_DIFF : REAL := 10.0;
	C : REAL := 1.33;
	H : REAL := 3.0;
END_VAR
VAR_OUTPUT
	TY : REAL;
	HEAT : BOOL;
END_VAR
VAR
	tr : REAL;
	tx: REAL;
END_VAR

(*
version 1.2	13. mar. 2009
programmer 	hugo
tested by		oscat

Heat_Temp calculates a heat characteristic based on the formula: tv=ti+(tvmax-ti)*((ti-tau)/(ti-taumin))^(1/n)
while
tv necessary heating temperature.
ti internal room temperature (20°C)
tau current external temperature
taumin external temperature to determine characteristics
C exponent for heating system (normally 1,33 or 1,1 for floor heating)

The two additional inputs TY_min and TY_max set limits for the output TY, while an offset inputs allows to rise or lower the room temperature.

*)

tr := T_INT + OFFSET;
tx := (tr - T_EXT) / (T_INT_CONFIG - T_EXT_CONFIG);

IF T_EXT + H > tr THEN
	TY := 0.0;
ELSE
	TY := LIMIT(TY_MIN, tr + T_DIFF * 0.5 * tx + (TY_CONFIG - T_DIFF * 0.5 - tr) * EXPT(tx, 1.0 / C), TY_MAX);
END_IF;

TY := MAX(TY, T_REQ);
HEAT := TY > 0.0;


(*

tv=ti+(tvmax-ti)*((ti-tau)/(ti-taumin))^(1/n)

tv aktuelle Vorlauftemp.
ti Raumtemperatur innen (20°C)
tau aktuelle Außentemperatur
taumin minimale Außentemperatur -12°C oder -15°C
n Heizkörperexponent (meistens 1,33)
Fußbodenheizung = 1,1
Wandheizung 1,3

Normen z. B. DIN 4703, DIN 4725 oder die Literatur, z. B Recknagel Abschnitt 1.3.5.

*)


(* revision history
hm	27. jan. 2008	rev 1.0
	original version

hm	26. sep. 2008	rev 1.1
	moved T_INT from config to Input
	added config variable H
	corrected error in formula

hm	13. mar. 2009	rev 1.2
	improved code

*)

END_FUNCTION_BLOCK

// POUs/Time&Date/HOUR_OF_DT
FUNCTION HOUR_OF_DT : INT
VAR_INPUT
	XDT : DT;
END_VAR


(*
	version 1.0	6. jun. 2008
	programmer 	oscat
	tested BY	oscat

HOUR_OF_DT returns the current hour (hour of the day) of a DT variable

*)

HOUR_OF_DT := DWORD_TO_INT((DT_TO_DWORD(XDT) MOD 86400)/3600);


(* revision history
hm		6.9.2008	rev 1.0
	original version


*)

END_FUNCTION

// POUs/Network/HTML_DECODE
FUNCTION HTML_DECODE : STRING(255)
VAR_INPUT
	IN : STRING(255);
END_VAR
VAR
	pos : INT;
	end : INT;
	tmp : STRING(10);
	code : STRING(1);
END_VAR


(*
version 1.2		17. dec. 2008
programmer 		hugo
tested by		oscat

HTML_DECODE converts HTML coded characters to text. 
&amp; is replaced by & ("Ampersand")
&lt; is replaced by < ("lower than")
&gt; is replaced by > ("greater than")
&quot; is replaced by " ("Quote")
all other &names characters are replaced by their respective character codes.

*)

HTML_DECODE := IN;

(* docode characters encoded by character position *)
pos := FIND(HTML_DECODE, '&');
WHILE pos > 0 DO
	tmp := MID(HTML_DECODE, 2, pos + 1);
	IF tmp = '#x' OR tmp = '#X' THEN
		(* hexadecimal representation found *)
		tmp := MID(HTML_DECODE, 10, pos + 3);
		end := FIND(tmp, ';');
		CODE := CHR_TO_STRING(DWORD_TO_BYTE(HEX_TO_DWORD(LEFT(tmp, end - 1))));
		HTML_DECODE := REPLACE(HTML_DECODE, CODE, end + 3, pos);
	ELSIF LEFT(tmp,1) = '#' THEN
		tmp := MID(HTML_DECODE, 10, pos + 2);
		end := FIND(tmp, ';');
		CODE := CHR_TO_STRING(INT_TO_BYTE(STRING_TO_INT(LEFT(tmp, end - 1))));
		HTML_DECODE := REPLACE(HTML_DECODE, CODE, end + 2, pos);
	ELSE
		(* replace all named characters *)
		tmp := MID(HTML_DECODE, 10, pos + 1);
		end := FIND(tmp, ';');
		CODE := CHR_TO_STRING(CHARCODE(LEFT(tmp, end - 1)));
		HTML_DECODE := REPLACE(HTML_DECODE, CODE, end + 1, pos);
	END_IF;
	(* search for next occurence of encoded characters *)
	pos := FINDP(HTML_DECODE, '&', pos + 1);
END_WHILE;



(* revision history
hm	3. mai. 2008	rev 1.0
	original version

hm	16. jun. 2008	rev 1.1
	changed nested call of replace for better compatibility

hm	17. dec. 2008	rev 1.2
	changed function CHR to CHR_TO_STRING

*)

END_FUNCTION

// POUs/Network/HTML_ENCODE
FUNCTION HTML_ENCODE : STRING(255)
VAR_INPUT
	IN : STRING(255);
	M : BOOL;
END_VAR
VAR
	pt_in : POINTER TO ARRAY[1..255] OF BYTE;
	pt_out : POINTER TO ARRAY[1..256] OF BYTE;
	pos_in : INT;
	pos_out : INT;
	stop : INT;
	B: BYTE;
	tmp : STRING(10);
	i: INT;
END_VAR


(*
version 1.0		3. mai. 2008
programmer 		hugo
tested by		hugo 

HTML_ENCODE checks a string if it contains reserved HTML characters and converts them to alternative html coding.
& is replaced by &amp; ("Ampersand")
< is replaced by &lt; ("lower than")
> is replaced by &gt; ("greater than")
" is replaced by &quot; ("Quote")

*)

pt_in  := ADR(in);
pt_out := ADR(HTML_ENCODE);

(* scan the input string and convert unallowed characters *)
pos_in := 1;
stop := LEN(in);
FOR pos_out := 1 TO 255 DO
	IF pos_in > stop THEN EXIT; END_IF;
	B := pt_in^[pos_in];
	CASE BYTE_TO_INT(B) OF
		34: (* " detected *)
			IF pos_out > 249 THEN EXIT; END_IF;
			pt_out^[pos_out] := 38;
			pos_out := pos_out + 1;
			pt_out^[pos_out] := 113;
			pos_out := pos_out + 1;
			pt_out^[pos_out] := 117;
			pos_out := pos_out + 1;
			pt_out^[pos_out] := 111;
			pos_out := pos_out + 1;
			pt_out^[pos_out] := 116;
			pos_out := pos_out + 1;
			pt_out^[pos_out] := 59;
		38: (* & detected *)
			IF pos_out > 250 THEN EXIT; END_IF;
			pt_out^[pos_out] := 38;
			pos_out := pos_out + 1;
			pt_out^[pos_out] := 97;
			pos_out := pos_out + 1;
			pt_out^[pos_out] := 109;
			pos_out := pos_out + 1;
			pt_out^[pos_out] := 112;
			pos_out := pos_out + 1;
			pt_out^[pos_out] := 59;
		60: (* < detected *)
			IF pos_out > 251 THEN EXIT; END_IF;
			pt_out^[pos_out] := 38;
			pos_out := pos_out + 1;
			pt_out^[pos_out] := 108;
			pos_out := pos_out + 1;
			pt_out^[pos_out] := 116;
			pos_out := pos_out + 1;
			pt_out^[pos_out] := 59;
		62: (* > detected *)
			IF pos_out > 251 THEN EXIT; END_IF;
			pt_out^[pos_out] := 38;
			pos_out := pos_out + 1;
			pt_out^[pos_out] := 103;
			pos_out := pos_out + 1;
			pt_out^[pos_out] := 116;
			pos_out := pos_out + 1;
			pt_out^[pos_out] := 59;
	ELSE
		IF M AND B > 127 THEN
			tmp := CHARNAME(B);
			(* exit if output string has not enough space *)
			IF pos_out + LEN(tmp) + 2 <= 255 THEN
				pt_out^[pos_out] := 38;
				pos_out := pos_out + 1;
				FOR i := 1 TO LEN(tmp) DO
					pt_out^[pos_out] := CODE(tmp, i);
					pos_out := pos_out + 1;
				END_FOR;
				pt_out^[pos_out] := 59;
			END_IF;
		ELSE
			pt_out^[pos_out] := B;
		END_IF;
	END_CASE;
	(* increment in by 1 *)
	pos_in := pos_in + 1;
END_FOR;

(* terminate the output string *)
pt_out^[pos_out] := 0;



(* revision history
hm		3. mai. 2008	rev 1.0
	original version

*)

END_FUNCTION

// POUs/Engineering/control/HYST
FUNCTION_BLOCK HYST
VAR_INPUT
	In : REAL;
	ON : REAL;
	OFF : REAL;
END_VAR
VAR_OUTPUT
	Q : BOOL;
	win : BOOL;
END_VAR


(*
version 1.0	2. jun. 2008
programmer 	hugo
tested BY	oscat

This Hystereses function has two modes:
1. if on > off then Q will be switched high when in > on and switched low when in < off.
2. if on < off then Q will be switched high when in < on and switched low when in > off.
the output win will be high when in is between low and high.

*)

IF ON >= OFF THEN
	IF IN < OFF THEN
		Q := FALSE;
		WIN := FALSE;
	ELSIF  IN > ON THEN
		Q := TRUE;
		WIN := FALSE;
	ELSE
		WIN := TRUE;
	END_IF;
ELSE
	IF IN > OFF THEN
		Q := FALSE;
		WIN := FALSE;
	ELSIF  IN < ON THEN
		Q := TRUE;
		WIN := FALSE;
	ELSE
		WIN := TRUE;
	END_IF;
END_IF;


(* revision history
hm		2.  jun 2008	rev 1.0
	original version

*)

END_FUNCTION_BLOCK

// POUs/Engineering/control/HYST_1
FUNCTION_BLOCK HYST_1
VAR_INPUT
	In : REAL;
	high : REAL;
	low : REAL;
END_VAR
VAR_OUTPUT
	Q : BOOL;
	win : BOOL;
END_VAR


(*
version 1.1	2. jun. 2008
programmer 	hugo
tested BY	oscat

this hysteresis function switches the output high if the input signal reaches obove high and will switch to low when the input falls back below low value.
a separate output mid is set if the input stays between low and high value.

*)

IF in < low THEN
	Q := FALSE;
	win := FALSE;
ELSIF in > high THEN
	Q := TRUE;
	win := FALSE;
ELSE
	win := TRUE;
END_IF;




(* revision history
hm		4.  aug. 2006	rev 1.0
	original version

hm		2. jun. 2008	rev 1.1
	improved performance
*)

END_FUNCTION_BLOCK

// POUs/Engineering/control/HYST_2
FUNCTION_BLOCK HYST_2
VAR_INPUT
	IN : REAL;
	VAL : REAL;
	HYS : REAL;
END_VAR
VAR_OUTPUT
	Q : BOOL;
	WIN: BOOL;
END_VAR
VAR
	tmp: REAL;
END_VAR


(*
version 1.2	2. jun. 2008
programmer 	oscat
tested BY	oscat

this hysteresis function switches the output high if the input signal reaches obove val + hys/2 and will switch to low when the input falls back below val - hys/2 value.
a separate output mid is set if the input stays between low and high value.

*)

tmp := val - hys * 0.5;
IF in < tmp THEN
	Q := FALSE;
	win := FALSE;
ELSIF in > tmp + hys THEN
	Q := TRUE;
	win := FALSE;
ELSE
	win := TRUE;
END_IF;



(* revision history
hm		4. aug 2006	rev 1.0
	original version

hm		5. jan 2008	rev 1.1
	improved code for better performance

hm		2. jun. 2008	rev 1.2
	improved performance
*)

END_FUNCTION_BLOCK

// POUs/Engineering/control/HYST_3
FUNCTION_BLOCK HYST_3
VAR_INPUT
	in : REAL;
	hyst : REAL;
	val1 : REAL;
	val2 : REAL;
END_VAR
VAR_OUTPUT
	Q1 : BOOL;
	Q2 : BOOL;
END_VAR
VAR
	X: REAL;
END_VAR

(*
version 1.2	5 jan 2008
programmer 	oscat
tested BY	oscat

this is a double hysteresis function. Out1 follows a hysteresis function defined by val1and hyst, while out 2 follows val2 and hyst.
if the input signal is between the two hysteresis switches (val1 and val2) then non of the outputs is active.

*)

X := hyst * 0.5;
IF in < val1 - X THEN
	q1 := TRUE;
ELSIF in > val1 + X THEN
	q1 := FALSE;
END_IF;
IF in < val2 - X THEN
	q2 := FALSE;
ELSIF in > val2 + X THEN
	q2 := TRUE;
END_IF;



(* revision history
hm	22. jan 2007	rev 1.0
	original version

hm	27. dec 2007	rev 1.1
	changed code for better performance

hm	5. jan 2008	rev 1.2
	further performance iprovements

*)

END_FUNCTION_BLOCK

// POUs/Engineering/automation/INC_DEC
FUNCTION_BLOCK INC_DEC
VAR_INPUT
	CHa : BOOL;
	CHb : BOOL;
	RST : BOOL;
END_VAR
VAR_OUTPUT
	dir : BOOL;
	cnt : INT;
END_VAR
VAR
	edgea : BOOL;
	clk: BOOL;
	clka: BOOL;
	clkb: BOOL;
	edgeb: BOOL;
	axb: BOOL;
END_VAR

(*
	version 1.0	4 aug 2006
	programmer 	oscat
	tested BY		oscat

incremental decoder with quadruple accuracy.
2 pulses for each channel are created for each directional pulse.
*)

axb := cha XOR chb;

(* create pulses for channel a *)
clka := cha XOR edgea;
edgea := cha;

clkb := chb XOR edgeb;
edgeb := chb;

(* create pulses for both channels *)
clk := clka OR clkb;

(* set the direction output *)
IF axb AND clka THEN dir := TRUE; END_IF;
IF axb AND clkb THEN dir := FALSE; END_IF;

(* increment or decrement the counter *)
IF clk AND dir THEN cnt := cnt + 1; END_IF;
IF clk AND NOT dir THEN cnt := cnt -1; END_IF;

(* reset the counter if rst active *)
IF rst THEN cnt := 0; END_IF;

END_FUNCTION_BLOCK

// POUs/Mathematical/INC2
FUNCTION INC2 : INT
VAR_INPUT
	X : INT;
	D : INT;
	L : INT;
	U : INT;
END_VAR
VAR
	tmp: INT;
END_VAR


(*
version 1.0	29. jun. 2008
programmer 	hugo
tested by	oscat

This function increments the input X by the value D and compares the result with U.
if the output exceeds U it will continue to count from L again.

*)

tmp := U - L + 1;
INC2 := (X + D - L + tmp) MOD tmp + L;



(* revision history
hm	29. jun. 2008		REV 1.0
	original version


*)

END_FUNCTION

// POUs/Logic/gate logic/INT_TO_BCDC
FUNCTION INT_TO_BCDC : BYTE
VAR_INPUT
	IN : INT;
END_VAR


(*
version 1.1	30. jun. 2008
programmer 	hugo
tested by		tobias

this function converts an integer into a two digit bcd number.
*)

INT_TO_BCDC := SHL(INT_TO_BYTE(IN / INT#10),4) OR INT_TO_BYTE(in MOD INT#10);

(* revision history
hm	13.12.2007
	original version

hm	30.6.2008	rev 1.1
	changed name INT_TO_BCD to INT_TO_BCDC to avoid collision with util.lib
	corrected error in code

*)

END_FUNCTION

// POUs/Engineering/automation/INTERLOCK_4
FUNCTION_BLOCK INTERLOCK_4
VAR_INPUT CONSTANT
END_VAR
VAR_INPUT
	I0 : BOOL;
	I1 : BOOL;
	I2 : BOOL;
	I3 : BOOL;
	E : BOOL;
	MODE : INT;

END_VAR
VAR_OUTPUT
	OUT : BYTE;
	TP : BOOL;
END_VAR
VAR
	in: BYTE;
	last: BYTE;
	old: BYTE;
	lmode: INT;
END_VAR

(*
version 1.1	14. mar. 2009
programmer 	hugo
tested by		oscat

INTERLOCK_4 detects one of 4 switches and delivers the number of the switch pressed on the output out
a output tp is true for one cycle if the output has changed.
a setup variable MODE selects between 3 different modes:
MODE = 0, any input active will disable all other inputs
MODE = 1, the input with the highest number will be acepted
mode = 2, the input last pressed will disable all others 

*)

(* check if enable is active *)
IF E THEN
(* reset all vars when there is a mode change on thy fly *)
	IF mode <> lmode THEN
		out := 0;
		last := 0;
		old := 0;
		lmode := mode;
	END_IF;
	(* load inputs into in *)
	in.0 := I0;
	in.1 := I1;
	in.2 := I2;
	in.3 := I3;
	(* only execute when there is any change *)
	IF in <> last THEN
		(* only execute when inputs have chages state *)
		CASE mode OF
			0:	(* output directly display inputs as bits in byte out *)
				out := in;

			1:	(* the input with the highest number will be acepted *)
				IF in.3 THEN out := 8;
				ELSIF in.2 THEN out := 4;
				ELSIF in.1 THEN out := 2;
				ELSE out := in;
				END_IF;

			2:	(* input last pressed will be displayed only *)
				last := ((in XOR last) AND in);
				IF last.3 THEN out := 8;
				ELSIF last.2 THEN out := 4;
				ELSIF last.1 THEN out := 2;
				ELSE out := last;
				END_IF;

			3:	(* any input active will disable all other inputs *)
				IF (out AND in) = 0 THEN
					IF in.3 THEN out := 8;
					ELSIF in.2 THEN out := 4;
					ELSIF in.1 THEN out := 2;
					ELSE out := in;
					END_IF;
				END_IF;

		END_CASE;
		last := in;
	END_IF;
	tp := out <> old;
	old := out;
ELSE
	out := 0;
	last := 0;
	old := 0;
	lmode := 0;
	tp := FALSE;
END_IF;


(* revision history
hm	24. oct 2008	rev 1.0
	original version

hm	14. mar. 2009	rev 1.1
	replaced double assignments

*)

END_FUNCTION_BLOCK

// POUs/Network/IP4_CHECK
FUNCTION IP4_CHECK : BOOL
VAR_INPUT
	NIP : DWORD;
	LIP : DWORD;
	SM : DWORD;
END_VAR


(*
version 1.0	4. mar 2008
programmer 	hugo
tested by		oscat

IP4_CHECK testet ob eine Network IP und Local_IP im selben Subnet sind.

*)

IP4_CHECK := (NIP AND sm) = (LIP AND SM);


(* revision history
hm		4. mar 2008	rev 1.0
	original version

*)

END_FUNCTION

// POUs/Network/IP4_DECODE
FUNCTION IP4_DECODE : DWORD
VAR_INPUT
	str : STRING(15);
END_VAR
VAR
	pos: INT;
END_VAR

(*
version 1.1	10. mar 2009
programmer 	kurt
tested by		hugo

IP4_DECODE testet ob ein string eine gültige IPv4 Adresse enthält und gibt die 4 Bytes der IP Adresse als DWORD zurück.

*)

pos := FIND(str, '.');
WHILE pos > 0 DO
	IP4_DECODE := SHL(IP4_DECODE,8) OR STRING_TO_DWORD(LEFT(str,pos - 1));
	str := DELETE(str, pos, 1);
	pos := FIND(str, '.');
END_WHILE;
IP4_DECODE := SHL(IP4_DECODE,8) OR STRING_TO_DWORD(str);


(* revision history
hm		29. feb 2008	rev 1.0
	original version

hm	10. mar. 2009	rev 1.1
	new algorythm
*)

END_FUNCTION

// POUs/Network/IP4_TO_STRING
FUNCTION IP4_TO_STRING : STRING(15)
VAR_INPUT
	IP4 : DWORD;
END_VAR
VAR
	tmp : STRING(3);
END_VAR

(*
version 1.1	10. mar. 2009
programmer 	kurt
tested by		hugo

IP4_TO_STRING erzeugt eine IP Adresse als String aus einem DWORD..

*)

(* mask bits AND INSERT AT given position *)
tmp := BYTE_TO_STRING(DWORD_TO_BYTE(IP4));
IP4_TO_STRING := CONCAT('...', tmp);
tmp := BYTE_TO_STRING(DWORD_TO_BYTE(SHR(IP4,8)));
IP4_TO_STRING := INSERT(IP4_TO_STRING, tmp, 2);
tmp := BYTE_TO_STRING(DWORD_TO_BYTE(SHR(IP4,16)));
IP4_TO_STRING := INSERT(IP4_TO_STRING, tmp, 1);
tmp := BYTE_TO_STRING(DWORD_TO_BYTE(SHR(IP4,24)));
IP4_TO_STRING := CONCAT(tmp, IP4_TO_STRING);



(* revision history
hm	22. apr 2008	rev 1.0
	original version

hm	10. mar. 2009	rev 1.1
	improved code
*)

END_FUNCTION

// POUs/Device Drivers/IRTRANS_1
FUNCTION_BLOCK IRTRANS_1
VAR_INPUT CONSTANT
	DEV_CODE : STRING;
	KEY_CODE : STRING;
END_VAR
VAR_INPUT
	CMD : BOOL;
END_VAR
VAR_IN_OUT
	DEV : STRING;
	KEY : STRING;
END_VAR
VAR_OUTPUT
	Q : BOOL;
END_VAR


(*
version 1.2	19. oct. 2008
programmer 	hugo
tested BY	oscat

*)

Q := cmd AND dev_code = dev AND key_code = key;

(* revision history
hm	2. jan 2008		rev 1.0
	original version

hm	20. 6. 2008		rev 1.1
	performance improvement

hm	19. oct. 2008	rev 1.2
	changed input device_code to dev_code and device to dev for compatibility reasons

*)

END_FUNCTION_BLOCK

// POUs/Device Drivers/IRTRANS_4
FUNCTION_BLOCK IRTRANS_4
VAR_INPUT CONSTANT
	DEV_CODE : STRING;
	KEY_CODE_0 : STRING;
	KEY_CODE_1 : STRING;
	KEY_CODE_2 : STRING;
	KEY_CODE_3 : STRING;
END_VAR
VAR_INPUT
	CMD : BOOL;
END_VAR
VAR_IN_OUT
	DEV : STRING;
	KEY : STRING;
END_VAR
VAR_OUTPUT
	Q0, Q1, Q2, Q3 : BOOL;
END_VAR
VAR
	decode: BOOL;
END_VAR

(*
version 1.2	19. oct. 2008
programmer 	hugo
tested BY	oscat

*)

decode := cmd AND dev_code = dev;

Q0 := key = key_code_0 AND decode;
Q1 := key = key_code_1 AND decode;
Q2 := key = key_code_2 AND decode;
Q3 := key = key_code_3 AND decode;



(* revision history
hm	2. jan 2008		rev 1.0
	original version

hm	17. oct. 2008	rev 1.1
	improved performance

hm	19. oct. 2008	rev 1.2
	changed input device_code to dev_code and device to dev for compatibility reasons
*)

END_FUNCTION_BLOCK

// POUs/Device Drivers/IRTRANS_8
FUNCTION_BLOCK IRTRANS_8
VAR_INPUT CONSTANT
	dev_code : STRING;
	key_code_0 : STRING;
	key_code_1 : STRING;
	key_code_2 : STRING;
	key_code_3 : STRING;
	key_code_4 : STRING;
	key_code_5 : STRING;
	key_code_6 : STRING;
	key_code_7 : STRING;
END_VAR
VAR_INPUT
	CMD : BOOL;
END_VAR
VAR_IN_OUT
	DEV : STRING;
	KEY : STRING;
END_VAR
VAR_OUTPUT
	Q0, Q1, Q2, Q3, Q4, Q5, Q6, Q7 : BOOL;
END_VAR
VAR
	decode: BOOL;
END_VAR

(*
version 1.2	19. oct. 2008
programmer 	hugo
tested BY	oscat

*)

decode := cmd AND dev_code = dev;

Q0 := key = key_code_0 AND decode;
Q1 := key = key_code_1 AND decode;
Q2 := key = key_code_2 AND decode;
Q3 := key = key_code_3 AND decode;
Q4 := key = key_code_4 AND decode;
Q5 := key = key_code_5 AND decode;
Q6 := key = key_code_6 AND decode;
Q7 := key = key_code_7 AND decode;


(* revision history
hm	2. jan 2008		rev 1.0
	original version

hm	17. oct 2008	rev 1.1
	improved performance

hm	19. oct. 2008	rev 1.2
	changed input device_code to dev_code and device to dev for compatibility reasons

*)

END_FUNCTION_BLOCK

// POUs/Device Drivers/IRTRANS_DECODE
FUNCTION_BLOCK IRTRANS_DECODE
VAR_INPUT
	BUFFER : POINTER TO ARRAY[0..32000] OF BYTE;
END_VAR
VAR_IN_OUT
	LENGTH : DINT;
END_VAR
VAR_OUTPUT
	CMD : BOOL;
	DEV : STRING;
	KEY : STRING;
	ERROR : BOOL;
END_VAR
VAR
	pt : POINTER TO BYTE;
	i : INT;
	stop : INT;
END_VAR

(*
version 1.1	19. oct. 2008
programmer 	hugo
tested BY	tobias

*)

(* do nothing if the buffer is empty *)
IF DINT_TO_INT(length) > 0 THEN
	i := 0;
	error := TRUE;
	stop := DINT_TO_INT(length) - 2;
	(* read characters before first comma and store in device *)
	pt := ADR(dev);
	WHILE i < stop DO
		IF buffer^[i] = 44 THEN EXIT; END_IF;
		pt^ := buffer^[i];
		pt := pt + 1;
		i := i + 1;
	END_WHILE;
	(* terminate the device string *)
	pt^ := 0;
	(* read after first comma and store in key *)
	i := i + 1;
	pt := ADR(key);
	WHILE i < stop DO
		pt^ := buffer^[i];
		pt := pt + 1;
		i := i + 1;
	END_WHILE;
	(* terminate the key string *)
	pt^:= 0;
	(* check if last two characters are $R$N 13, 10 *)
	IF buffer^[i] <> 13 AND buffer^[i+1] <> 10 THEN	RETURN;	END_IF;
	(* check if device and key are present *)
	IF LEN(dev) = 0 OR LEN(key) = 0 THEN RETURN; END_IF;
	(* a valid transmission has been received *)
	cmd := TRUE;
	error := FALSE;
	(* clear the input buffer to allow the next transmission to occur *)
	length := 0;
ELSE
	error := FALSE;
	cmd := FALSE;
END_IF;


(* revision history
hm	2. jan 2008		rev 1.0
	original version

hm	19. oct. 2008	rev 1.1
	added typecast to avoid warnings
	changed output device to dev for compatibility reasons

*)

END_FUNCTION_BLOCK

// POUs/String/IS_ALNUM
FUNCTION IS_ALNUM : BOOL
VAR_INPUT
	str : STRING(STRING_LENGTH);
END_VAR
VAR
	L: INT;
	pt : POINTER TO BYTE;
	pos: INT;
END_VAR

(*
version 1.1	29. mar. 2008
programmer 		kurt
tested by		hugo

ISC_ALNUM testet ob in einem string nur Zahlen 0..9 vorkommen.

*)

PT := ADR(str);
L := LEN(str);
FOR pos := 1 TO L DO
	IF NOT (ISC_ALPHA(pt^) OR ISC_NUM(pt^)) THEN
		IS_ALNUM := FALSE;
		RETURN;
	END_IF;
    	PT := PT + 1;
END_FOR;
IS_ALNUM := L > 0;


(* revision history
hm	29. feb 2008	rev 1.0
	original version

hm	29. mar. 2008	rev 1.1
	changed STRING to STRING(STRING_LENGTH)
*)

END_FUNCTION

// POUs/String/ISC_ALPHA
FUNCTION ISC_ALPHA : BOOL
VAR_INPUT
	IN : BYTE;
END_VAR


(*
version 1.1	19. oct. 2008
programmer 	oscat
tested by	oscat

ISC_ALPHA checks if a character is a..z or A..Z.

*)

IF setup.EXTENDED_ASCII THEN
	ISC_ALPHA := (in > 64 AND in < 91) OR (in > 191  AND in <> 215 AND in <> 247) OR (in > 96 AND in < 123);
ELSE
	ISC_ALPHA := (IN > 64 AND IN < 91) OR (in > 96 AND in < 123);
END_IF;

(* revision history
hm	6. mar. 2008	rev 1.0
	original version

hm	19. oct. 2008	rev 1.1
	changes setup constants
*)

END_FUNCTION

// POUs/String/ISC_NUM
FUNCTION ISC_NUM : BOOL
VAR_INPUT
	IN : BYTE;
END_VAR


(*
version 1.0	6. mar 2008
programmer 	oscat
tested by		hugo

ISC_NUM checks if a character is 0..9.

*)

ISC_NUM := IN > 47 AND IN < 58;

(* revision history
hm		6. mar. 2008	rev 1.0
	original version

*)

END_FUNCTION

// POUs/String/IS_ALPHA
FUNCTION IS_ALPHA : BOOL
VAR_INPUT
	str : STRING(STRING_LENGTH);
END_VAR
VAR
	L: INT;
	pt : POINTER TO BYTE;
	pos: INT;
END_VAR

(*
version 1.1	29. mar. 2008
programmer 		kurt
tested by		hugo

IS_ALPHA testet ob in einem string nur Zeichen a-z oder A - Z vorkommen.

*)

PT := ADR(str);
L := LEN(str);
FOR pos := 1 TO L DO
	IF NOT ISC_ALPHA(pt^) THEN
		IS_ALPHA := FALSE;
		RETURN;
	END_IF;
    	PT := PT + 1;
END_FOR;
IS_ALPHA := L > 0;


(* revision history
hm	29. feb 2008	rev 1.0
	original version

hm	29. mar. 2008	rev 1.1
	changed STRING to STRING(STRING_LENGTH)
*)

END_FUNCTION

// POUs/String/IS_CC
FUNCTION IS_CC : BOOL
VAR_INPUT
	str : STRING(STRING_LENGTH);
	cmp : STRING(STRING_LENGTH);
END_VAR
VAR
	L: INT;
	pos: INT;
END_VAR

(*
version 1.1	29. mar. 2008
programmer 	Tobias
tested by	hugo

ISC_CC testet ob ein string nur aus Zeichen des Strings CMP besteht.

*)

L := LEN(str);
FOR pos := 1 TO L DO
	IF FIND(CMP,MID(str,1,pos)) = 0 THEN RETURN; END_IF;
END_FOR;
IS_CC := L > 0;



(* revision history
hm	19. mar 2008	rev 1.0
	original version

hm	29. mar. 2008	rev 1.1
	changed STRING to STRING(STRING_LENGTH)
*)

END_FUNCTION

// POUs/String/IS_CTRL
FUNCTION IS_CTRL : BOOL
VAR_INPUT
	STR : STRING(STRING_LENGTH);
END_VAR
VAR
	L: INT;
	pt : POINTER TO BYTE;
	pos: INT;
END_VAR

(*
version 1.1	29. mar 2008
programmer 		kurt
tested by		hugo

IS_CTRL testet ob in einem string nur Steuerzeichen (Char < 32) vorkommen.

*)

PT := ADR(str);
L := LEN(str);
FOR pos := 1 TO L DO
	IF NOT (ISC_CTRL(pt^)) THEN
		IS_CTRL := FALSE;
		RETURN;
	END_IF;
    	PT := PT + 1;
END_FOR;
IS_CTRL := L > 0;


(* revision history
hm	29. feb. 2008	rev 1.0
	original version

hm	29. mar. 2008	rev 1.1
	changed STRING to STRING(STRING_LENGTH)
*)

END_FUNCTION

// POUs/String/ISC_CTRL
FUNCTION ISC_CTRL : BOOL
VAR_INPUT
	IN : BYTE;
END_VAR


(*
version 1.0	6. mar 2008
programmer 	oscat
tested by		hugo

ISC_ALPHA checks if a character is a control character.

*)

ISC_CTRL := IN < 32 OR IN = 127;

(* revision history
hm		6. mar. 2008	rev 1.0
	original version

*)

END_FUNCTION

// POUs/String/IS_HEX
FUNCTION IS_HEX : BOOL
VAR_INPUT
	str : STRING(STRING_LENGTH);
END_VAR
VAR
	L: INT;
	pt : POINTER TO BYTE;
	pos: INT;
END_VAR

(*
version 1.1	29. mar. 2008
programmer 		kurt
tested by		hugo

IS_HEX testet ob in einem string nur Zahlen 0..9 oder A..F oder a..f  vorkommen.

*)

PT := ADR(str);
L := LEN(str);
FOR pos := 1 TO L DO
	IF NOT (ISC_HEX(pt^)) THEN
		IS_HEX := FALSE;
		RETURN;
	END_IF;
    	PT := PT + 1;
END_FOR;
IS_HEX := L > 0;


(* revision history
hm	29. feb 2008	rev 1.0
	original version

hm	29. mar. 2008	rev 1.1
	changed STRING to STRING(STRING_LENGTH)
*)

END_FUNCTION

// POUs/String/ISC_HEX
FUNCTION ISC_HEX : BOOL
VAR_INPUT
	IN : BYTE;
END_VAR


(*
version 1.0	6. mar 2008
programmer 	oscat
tested by		hugo

ISC_HEX checks if a character is 0..9, A..F, a..f.

*)

ISC_HEX := (IN > 47 AND IN < 58) OR (IN > 64 AND IN < 71) OR (IN > 96 AND IN < 103);

(* revision history
hm		6. mar. 2008	rev 1.0
	original version

*)

END_FUNCTION

// POUs/Network/IS_IP4
FUNCTION IS_IP4 : BOOL
VAR_INPUT
	str : STRING;
END_VAR


(*
version 1.1	10. mar 2009
programmer 	kurt
tested by		hugo

IS_IP4 testet ob ein string eine gültige IPv4 Adresse enthält.

*)

IS_IP4 := COUNT_CHAR(str, 46) = 3;


(* revision history
hm	1. mar. 2008	rev 1.0
	original version

hm	10. mar. 2009	rev 1.1
	new code

*)

END_FUNCTION

// POUs/String/IS_LOWER
FUNCTION IS_LOWER : BOOL
VAR_INPUT
	str : STRING(STRING_LENGTH);
END_VAR
VAR
	l: INT;
	pt : POINTER TO BYTE;
	pos: INT;
END_VAR

(*
version 1.1	29. mar. 2008
programmer 		kurt
tested by		hugo

IS_LOWER testet ob in einem string nur kleinbuchstaben vorkommen.

*)

PT := ADR(str);
L := LEN(str);
FOR pos := 1 TO L DO
	IF NOT (ISC_LOWER(pt^)) THEN
		IS_LOWER := FALSE;
		RETURN;
	END_IF;
    	PT := PT + 1;
END_FOR;
IS_LOWER := L > 0;


(* revision history
hm	29. feb 2008	rev 1.0
	original version

hm	29. mar. 2008	rev 1.1
	changed STRING to STRING(STRING_LENGTH)
*)

END_FUNCTION

// POUs/String/ISC_LOWER
FUNCTION ISC_LOWER : BOOL
VAR_INPUT
	IN : BYTE;
END_VAR


(*
version 1.1	19. oct. 2008
programmer 	hugo
tested by	oscat

isc_lower checks if a character is lowercase.

*)

IF setup.EXTENDED_ASCII THEN
	ISC_LOWER := ((in > 96) AND (in < 123)) OR ((in > 222) AND (in <> 247));
ELSE
	ISC_LOWER := ((in > 96) AND (in < 123));
END_IF;

(* revision history
hm	6. mar. 2008	rev 1.0
	original version

hm	19. oct. 2008	rev 1.1
	changes setup constants
*)

END_FUNCTION

// POUs/String/IS_NCC
FUNCTION IS_NCC : BOOL
VAR_INPUT
	str : STRING(STRING_LENGTH);
	cmp : STRING(STRING_LENGTH);
END_VAR
VAR
	L: INT;
	pos: INT;
END_VAR

(*
version 1.1	29. mar. 2008
programmer 	Tobias
tested by		hugo

IS_NCC testet ob in einem string keine Zeichen des Strings CMP enthalten sind.

*)

L := LEN(str);
FOR pos := 1 TO L DO
	IF FIND(CMP,MID(str,1,pos)) > 0 THEN RETURN; END_IF;
END_FOR;
IS_NCC := TRUE;



(* revision history
hm	19. mar 2008	rev 1.0
	original version

hm	29. mar. 2008	rev 1.1
	changed STRING to STRING(STRING_LENGTH)
*)

END_FUNCTION

// POUs/String/IS_NUM
FUNCTION IS_NUM : BOOL
VAR_INPUT
	str : STRING(STRING_LENGTH);
END_VAR
VAR
	L : INT;
	pt : POINTER TO BYTE;
	pos: INT;
END_VAR

(*
version 1.1	29. mar. 2008
programmer 		kurt
tested by		hugo

IS_NUM testet ob in einem string nur Zahlen 0..9 vorkommen.

*)

PT := ADR(str);
L := LEN(str);
FOR pos := 1 TO L DO
	IF NOT (ISC_NUM(pt^)) THEN
		IS_NUM := FALSE;
		RETURN;
	END_IF;
    	PT := PT + 1;
END_FOR;
IS_NUM := L > 0;


(* revision history
hm	29. feb 2008	rev 1.0
	original version

hm	29. mar. 2008	rev 1.1
	changed STRING to STRING(STRING_LENGTH)
*)

END_FUNCTION

// POUs/Mathematical/Array/IS_SORTED
FUNCTION IS_SORTED : BOOL
VAR_INPUT
	pt : POINTER TO ARRAY[0..32000] OF REAL;
	size : UINT;
END_VAR
VAR

	stop: INT;
	i: INT;
END_VAR

(*
version 1.1	4. apr. 2008
programmer 	hugo
tested by	tobias

this function will return true if the given array is sorted in an ascending order.
the function needs to be called:	array_sorted(adr("array"),sizeof("array"));
because this function works with pointers its very time efficient and it needs no extra memory.

*)

stop := UINT_TO_INT(SHR(size,2)-2);
FOR i := 0 TO stop DO
	IF pt^[i] > pt^[i+1] THEN
		IS_SORTED := FALSE;
		RETURN;
	END_IF;
END_FOR;

IS_SORTED := TRUE;

(* revision history

hm 	29. mar. 2008 	rev 1.0
	original version

hm	4. apr. 2008	rev 1.1
	added type conversion to avoid warnings under codesys 3.0
*)

END_FUNCTION

// POUs/String/IS_UPPER
FUNCTION IS_UPPER : BOOL
VAR_INPUT
	str : STRING(STRING_LENGTH);
END_VAR
VAR
	L: INT;
	pt : POINTER TO BYTE;
	pos: INT;
END_VAR

(*
version 1.1	29. mar. 2008
programmer 		kurt
tested by		hugo

IS_UPPER testet ob in einem string keine Kleinbuchstaben vorkommen.

*)

PT := ADR(str);
L := LEN(str);
FOR pos := 1 TO L DO
	IF NOT (ISC_UPPER(pt^)) THEN
		IS_UPPER := FALSE;
		RETURN;
	END_IF;
    	PT := PT + 1;
END_FOR;
IS_UPPER := L > 0;


(* revision history
hm	29. feb 2008	rev 1.0
	original version

hm	29. mar. 2008	rev 1.1
	changed STRING to STRING(STRING_LENGTH)
*)

END_FUNCTION

// POUs/String/ISC_UPPER
FUNCTION ISC_UPPER : BOOL
VAR_INPUT
	IN : BYTE;
END_VAR


(*
version 1.1	19. oct. 2008
programmer 	hugo
tested by	oscat

ISC_upper checks if a character is uppercase

*)

IF setup.EXTENDED_ASCII THEN
	ISC_UPPER :=  ((in > 64) AND (in < 91)) OR (((in > 191) AND (in < 223)) AND (in <> 215));
ELSE
	ISC_UPPER := ((in > 64) AND (in < 91));
END_IF;


(* revision history
hm	6. mar. 2008	rev 1.0
	original version

hm	19. oct. 2008	rev 1.1
	changes setup constants

*)

END_FUNCTION

// POUs/Network/IS_URLCHR
FUNCTION IS_URLCHR : BOOL
VAR_INPUT
	IN : BYTE;
END_VAR


(*
version 1.0		27. apr. 2008
programmer 		hugo
tested by		hugo

IS_URL_CHR is true if a string contains only non reserved characters for an url.
the non reserved characters are : [A..Z], [a..z], [0..9], -_.~

*)

IS_URLCHR := ((IN > 47) AND (IN < 58)) OR ((IN > 64) AND (IN < 91)) OR ((IN > 96) AND (IN < 123)) OR (in = 126) OR (in = 95) OR (in =45) OR (in =46);


(* revision history
hm		27. apr. 2008	rev 1.0
	original version

*)

END_FUNCTION

// POUs/Time&Date/JD2000
FUNCTION JD2000 : REAL
VAR_INPUT
	DTI : DT;
END_VAR


(*
version 1.0	15. jul. 2008
programmer 	hugo
tested by	oscat

JULIAN calculates the astronomic julian date.

*)

JD2000 := DWORD_TO_REAL(DT_TO_DWORD(DTI) - 946728000) / 86400.0;



(* revision histroy
hm	15. jul. 2008	rev 1.0
	original release


*)

END_FUNCTION

// POUs/Engineering/conversion/K_TO_C
FUNCTION K_TO_C : REAL
VAR_INPUT
	Kelvin : REAL;
END_VAR


(*
version 1.1	19. aug 2009
programmer 	hugo
tested by		tobias

this function converts kelvin to celsius

*)

K_TO_C := Kelvin + phys.T0;


(* revision history

hm	4. aug 2006	rev 1.0
	original version

hm	19. aug 2009	rev 1.1
	fixed calculation error

*)

END_FUNCTION

// POUs/Engineering/conversion/KMH_TO_MS
FUNCTION KMH_TO_MS : REAL
VAR_INPUT
	kmh : REAL;
END_VAR


(*
version 1.1	6 jan 2007
programmer 	hugo
tested by		tobias

this function converts velocities from Kilometers / hour to Meters / Second

*)

KMH_TO_MS := kmh * 0.2777777777777;

(* revision history
hm	4. feb 2007		rev 1.0
	original version

hm	6. jan 2008		rev 1.1
	improved performance

*)

END_FUNCTION

// POUs/Mathematical/LAMBERT_W
FUNCTION LAMBERT_W : REAL
VAR_INPUT
	X : REAL;
END_VAR
VAR
	w : REAL;
	i : INT;
	we: REAL;
	w1e: REAL;
	last: DWORD;
	ewx: REAL;
END_VAR



(*
version 1.1	10. mar. 2009
programmer 	hugo
tested by		oscat

this function calculates the lambert_w function.

*)

(* check for valid input and return -1000 if too low *)
IF x < -0.367879441171442 THEN
	LAMBERT_W := -1000.0;
	RETURN;
(* return 0 if x = 0 *)
ELSIF x = 0.0 THEN
	RETURN;
(* first an estimate is calculated *)
ELSIF x <= 500.0 THEN
	w := LN(x + 1.0);
	w := 0.665 * (1.0 + 0.0195 * w) * w + 0.04;
ELSE
	w := LN(x - 4.0) - (1.0 - 1.0/LN(x)) * LN(LN(x));
END_IF;
(* use estimate to calculate exact result *)
FOR i := 0 TO 5 DO
	ewx := EXP(w);
	we := w * ewx - x;
	w1e := (w+1.0) * ewx;
	last := REAL_TO_DW(w) AND 16#FFFF_FFFC;
	w := w - (we / (w1e - (w+2.0) * we / (2.0 * w + 2.0)));
	IF (REAL_TO_DW(w) AND 16#FFFF_FFFC) = last THEN EXIT; END_IF;
END_FOR;
LAMBERT_W := w;


(* revision hisdtory
hm	26. oct. 2008	rev 1.0
	original version

hm	10. mar. 2009	rev 1.1
	real constants updated to new systax using dot

*)

END_FUNCTION

// POUs/Logic/gate logic/REAL_TO_DW
FUNCTION REAL_TO_DW : DWORD
VAR_INPUT
	X : REAL;
END_VAR
VAR
	pt : POINTER TO DWORD;
END_VAR

(*
version 1.0	18. apr. 2008
programmer 	hugo
tested by		tobias

this function converts a 32 Bit Real to a dword in a bitwise manner.
*)

pt := ADR(X);
REAL_TO_DW := pt^;

(* revision history
hm	18. apr. 2008
	original version

*)

END_FUNCTION

// POUs/Mathematical/LANGEVIN
FUNCTION LANGEVIN : REAL
VAR_INPUT
	X : REAL;
END_VAR


(*
version 1.2	10.mar. 2009
programmer 	hugo
tested by		tobias

this function calculates the langevin function

*)

IF X = 0.0 THEN
	LANGEVIN := 0.0;
ELSE
	LANGEVIN := COTH(X) - 1.0 / X;
END_IF;

(* revision history
hm	10.12.2007	rev 1.0
	original version

hm	11. mar 2008	rev 1.1
	changed formula to avoid problems when x = 0

hm	10. mar. 2009	rev 1.2
	real constants updated to new systax using dot

*)

END_FUNCTION

// POUs/Time&Date/LEAP_DAY
FUNCTION LEAP_DAY : BOOL
VAR_INPUT
	IDATE : DATE;
END_VAR


(*
version 1.1	7. oct. 2008
programmer 	hugo
tested by	oscat


leap_day is true if the tested day is a leap day (29. of february).  
  
*)

LEAP_DAY := (MONTH_OF_DATE(idate) = 2) AND (DAY_OF_MONTH(idate) = 29);



(* change history

hm 	15. jun. 2008	rev 1.0
	original version

hm	7. oct. 2008	rev 1.1
	changed function month to month_of_date
*)

END_FUNCTION

// POUs/Building/HLK/LEGIONELLA
FUNCTION_BLOCK LEGIONELLA
VAR_INPUT
	manual : BOOL;
	temp_boiler : REAL;
	temp_return : REAL := 100.0;
	DT_in: DT;
	rst : BOOL;
END_VAR
VAR_INPUT CONSTANT
	T_start: TOD := tod#03:00:00;
	day : INT := 7;
	temp_set : REAL := 70.0;
	temp_offset : REAL := 10.0;
	temp_hys : REAL := 5.0;
	t_max_heat: TIME := t#10m;
	t_max_ret : TIME := t#10m;
	tp_0: TIME := t#5m;
	TP_1: TIME := t#5m;
	tp_2: TIME := t#5m;
	tp_3: TIME := t#5m;
	tp_4: TIME := t#5m;
	tp_5: TIME := t#5m;
	tp_6: TIME := t#5m;
	tp_7: TIME := t#5m;
END_VAR
VAR_OUTPUT
	Heat : BOOL;
	pump : BOOL;
	valve0 : BOOL;
	valve1 : BOOL;
	valve2 : BOOL;
	valve3 : BOOL;
	valve4 : BOOL;
	valve5 : BOOL;
	valve6 : BOOL;
	valve7 : BOOL;
	run: BOOL;
	Status : BYTE;
END_VAR
VAR
	X1: TIMER_1;
	x2: SEQUENCE_8;
	x3: HYST_1;
	init: BOOL;
END_VAR

(*
version 1.3	13. mar. 2009
programmer 	oscat
tested by		oscat

Legionella is a complete sequencer for up to 8 hot water lines that need to be sterilzed periodically.
legionella needs a DT input with the appropriate time, usually gererated by the rtc of the system. for system independence this time is connected externally.
T_start is the time when sterilazation should be started and day is the day_of_week when it should be performed (1=Monday and 7=sunday).
so sterilazation is autioimatically performed once a week at a specified time.
temp_set and temp_hys and temp_offset specify the boiler temperatur nedded for sterilization. as a defaut Temp_set is set to 70 deg C and Temp_hys is set to 5 deg C and temp_offset is 10 deg C.
a temp boiler input reads the boiler temperature of the hot water tank.
after a start pulse is gererated by the weekly timer or a manual test input the sequence is started:
1. the boiler is heated to temp_set + temp_offset + temp_hys = 85 deg C unless chaged at setup.
	the heat output is turned on and tells the heater to turn heating on. if the temp is not reached for a time of t_max_heat (10 min) the error output is set and the sequence is stopped.
2. after the specified temperature is reached, the output valve0 and pump is turned on and starts sterilization of line0 until temp_return has reached temp_set and continues to sterilize for a time of tp_0 (5 min default).
	if tmep_set is not reached at the temp_return_input then the error output is set and the sequence will be stopped.
	if there is no temp sensor for temp_return (the temperature at the return point for the circulation pump pls set this imput to a value greater then temp_set (by default use 100 deg C).
	in this case sterilization is performed for the default times without monitoring the return temp.
3. this sequence is repeated for up to valves.

connection scheme:

temp_boiler:	input oif the boiler temperature sensor.
temp_hys:		config value for the heater hysteresis, preset to 5 deg C.
temp_offset:	config value for the heater temp_offset against temp_set, preset to 10 deg C.
temp_set:		config value for the specified sterilization temperature, preset to 70 deg C.
temp_return:	input of the circulation return line temperature sensor, if not availabe set this value to 100 deg C.
manual:		manual input to start the sterilization by hand for diagnostic purposes, rising edge active, leave low for automatic operation.
DT_in:			date,time input supplied by a external real time clock.
T_start:		time of day when the sterilization should be started.
day:			config value for day of week when the process should be started, preset to sunday.
t_max_hest:	tmax time to be needed for the heater to heat the hot water tank to the specified value, preset to 10 min.

*)

(* startup initialization *)
IF NOT init THEN
	init := TRUE;
	X1.day := SHR(BYTE#128,day);
	X1.start := T_start;
	X3.low := Temp_offset + temp_set;
	X3.high := Temp_hys + X3.low;
	X2.wait0 := T_max_heat;
	X2.delay0 := TP_0;
	X2.delay1 := TP_1;
	X2.delay2 := TP_2;
	X2.delay3 := TP_3;
	X2.delay4 := TP_4;
	X2.delay5 := TP_5;
	X2.delay6 := TP_6;
	X2.delay7 := TP_7;
	X2.wait1 := T_max_ret;
	X2.wait2 := T_max_ret;
	X2.wait3 := T_max_ret;
	X2.wait4 := T_max_ret;
	X2.wait5 := T_max_ret;
	X2.wait6 := T_max_ret;
	X2.wait7 := T_max_ret;
	X2();
END_IF;

(* oerational code *)
X1(DTi := DT_in);
IF X1.Q OR MANUAL OR x2.run THEN
	X3(in := temp_boiler);
	X2.in0 := X3.Q OR x3.win;
	X2.in1 := temp_return >= temp_set;
	X2.in2 := x2.in1;
	X2.in3 := x2.in1;
	X2.in4 := x2.in1;
	X2.in5 := x2.in1;
	X2.in6 := x2.in1;
	X2.in7 := x2.in1;
	X2.rst := rst;
	X2(start := X1.Q OR MANUAL);
	run := x2.run;
	pump := x2.qx;
	Heat := NOT X3.Q AND x2.run;
	valve0 := X2.Q0;
	valve1 := X2.Q1;
	valve2 := X2.Q2;
	valve3 := X2.Q3;
	valve4 := X2.Q4;
	valve5 := X2.Q5;
	valve6 := X2.Q6;
	valve7 := X2.Q7;
	pump := X2.qx;
	status := X2.status;
ELSE;
	X2(start :=0);
	status := x2.status;
END_IF;

(* revision history

hm 17.jan 2007	rev 1.1
	rewritten to st for higher performance
	changes eeror output to esr compatible status output

hm	23. 10.2008	rev 1.2
	update code to use new version of timer_1

hm	13. mar. 2009	rev 1.3
	real constants updated to new systax using dot
	using new module sequence_8
*)

END_FUNCTION_BLOCK

// POUs/Logic/generators/TP_1
FUNCTION_BLOCK TP_1
VAR_INPUT
	IN : BOOL;
	PT : TIME;
	RST : BOOL;
END_VAR
VAR_OUTPUT
	Q : BOOL;
END_VAR
VAR
	tx : TIME;
	start : TIME;
	ix : BOOL;
END_VAR

(*
version 1.0	28. jun. 2008
programmer 	hugo
tested by		oscat

TP_1 generates a pulse every time it is calles with in := TRUE.
in addition the timer can be cleared asynchronously with rst.
the timer can be retriggered as often as necessary. it will count PT from the last trigger.

*)

(* read system timer *)
tx := DWORD_TO_TIME(T_PLC_MS());

IF RST THEN
	Q := FALSE;
ELSIF IN AND NOT ix THEN
	Q := TRUE;
	start := tx;
ELSIF tx - start >= PT THEN
	Q := FALSE;
END_IF;

ix:= IN;



(* revision history
hm	28. jun. 2008
	original version

*)

END_FUNCTION_BLOCK

// POUs/Building/electrical/TIMER_1
FUNCTION_BLOCK TIMER_1
VAR_INPUT
	E : BOOL := TRUE;
	DTI : DT;
	START : TOD;
	DURATION : TIME;
	DAY : BYTE := 2#0111_1111;
END_VAR
VAR_OUTPUT
	Q : BOOL;
END_VAR
VAR
	td : DATE;
	tdt : DT;
END_VAR

(*
version 2.1	6. nov. 2008
programmer 	oscat
tested by	oscat

this is a simple timer that generates an output pulse on selected days.
the output pulse width can be programmed with duration, if set to 0 no pulse is generated.
day specifies the specific days for the event to occur, bit 0 = sunday, bit 1 = saturday, bit 2 = friday ....
for all days to be active 127 has to be specified for DAY.

*)

td := DT_TO_DATE(DTI);
tdt := DATE_TO_DT(td) + TOD_TO_TIME(start);

Q := DTI >= tdt AND dti < tdt + duration AND E AND (SHR(BYTE#128, DAY_OF_WEEK(td)) AND day) > 0;



(*
1.12.2006 hm		rev 1.1
	corrected an error with pulse width = 0.

25.12.2006 hm		rev 1.2
	corrected an error when timer overflows.

14.apr 2007 hm		rev 1.3
	corrected an error while while output would not go active when start year would be 1970.
	increase accuracy by checking every 100ms
	added init section to compensate for timer overflow

15.9.2007 hm		rev 1.4
	replaced Time() with T_PLC_MS for compatibility and performance reasons

hm	1. okt 2007		rev 1.5
	corrected an error while output would not stay active over midnight.

hm	17. jan 2008	rev 1.6
	New code with better performance  
	Output is now only active during the time of day it is supposed to 
	no pulse is generated at power up

hm	7. oct. 2008	rev 1.7
	changed function weekday to day_of_week

hm	23. oct. 2008	rev 2.0
	new code, added input E, now days can be selected by bits in byte day

hm	6. nov. 2008	rev 2.1
	added default for input EN and input DAY
*)

END_FUNCTION_BLOCK

// POUs/Logic/generators/SEQUENCE_8
FUNCTION_BLOCK SEQUENCE_8
VAR_INPUT
	in0 : BOOL := TRUE;
	in1 : BOOL := TRUE;
	in2 : BOOL := TRUE;
	in3 : BOOL := TRUE;
	in4 : BOOL := TRUE;
	in5 : BOOL := TRUE;
	in6 : BOOL := TRUE;
	in7 : BOOL := TRUE;
	start : BOOL;
	rst : BOOL;
	wait0 : TIME;
	delay0 : TIME;
	wait1 : TIME;
	delay1 : TIME;
	wait2 : TIME;
	delay2 : TIME;
	wait3 : TIME;
	delay3 : TIME;
	wait4 : TIME;
	delay4 : TIME;
	wait5 : TIME;
	delay5 : TIME;
	wait6 : TIME;
	delay6 : TIME;
	wait7 : TIME;
	delay7 : TIME;
END_VAR
VAR_INPUT CONSTANT
	stop_on_error : BOOL;
END_VAR
VAR_OUTPUT
	Q0 : BOOL;
	Q1 : BOOL;
	Q2 : BOOL;
	Q3 : BOOL;
	Q4 : BOOL;
	Q5 : BOOL;
	Q6 : BOOL;
	Q7 : BOOL;
	QX : BOOL;
	run: BOOL;
	step : INT := -1;
	status : BYTE;
END_VAR
VAR
	last : TIME;
	edge : BOOL;
	tx: TIME;
	init: BOOL;
END_VAR

(*
version 1.5	13. mar. 2009
programmer 	oscat
tested by		hans

sequence_8 enables run when a low to high transition is present on start.
a low to high transition on start will restart the sequencer at any time while a rst will hold the sequencer in reset while true.
after run is enabled with a rising edge on start the sequencer waits for wait0 on in0 to enable q0 which stays on for delay0.
the next cycle starts with wait1, continues with delay 1 and so on...
if an edge is not detected during the wait period, the sequencer will then display the error number on the status output.
The status numbers are 1 .. 8 for erros in step 0..7.
after the last step that sets q7, the sequencer leaves q7 on for delay7 and then resets to the initial state.
a step output will indicate the current step of the sequencer and will also be present with a fault condition.
after the first output is turened on the sequencer switches from q0 to q1 and so on, at any time there is only one output enabled.
if an input signal is not detected during a wait period, the sequencer will display the error number ( 1 for in0, 2 for in1 .... ).
when an error is present and the config variable stop_on_error is set then the sequencer will stop. otherwise it will continue.
The status output will also display 110 for waiting and 111 sequece running.

*)

(* read sps timer *)
tx := DWORD_TO_TIME(T_PLC_MS());

(* initialize on startup *)
IF NOT init THEN
	last := tx;
	init := TRUE;
	status := 110;
END_IF;

(* asynchronous reset *)
IF rst THEN
	step := -1;
	Q0 := 0;
	Q1 := 0;
	Q2 := 0;
	Q3 := 0;
	Q4 := 0;
	Q5 := 0;
	Q6 := 0;
	Q7 := 0;
	status := 110;
	run := 0;

(* edge on start input restarts the sequencer *)
ELSIF start AND NOT edge THEN
	step := 0;
	last := tx;
	status := 111;
	Q0 := 0;
	Q1 := 0;
	Q2 := 0;
	Q3 := 0;
	Q4 := 0;
	Q5 := 0;
	Q6 := 0;
	Q7 := 0;
	run := 1;
END_IF;
edge := start;

(* check if stop on error is necessary *)
IF status > 0 AND status < 100 AND stop_on_error THEN RETURN; END_IF;

(* sequence is running *)
IF run AND step = 0 THEN
	IF NOT q0 AND in0 AND tx - last <= wait0 THEN
		Q0 := TRUE;
		last := tx;
	ELSIF NOT q0 AND tx - last > wait0 THEN
		status := 1;
		run := FALSE;
	ELSIF q0 AND tx - last >= delay0 THEN
		step := 1;
		last := tx;
	END_IF;
END_IF;
IF run AND step = 1 THEN
	IF NOT q1 AND in1 AND tx - last <= wait1 THEN
		Q0 := FALSE;
		Q1 := TRUE;
		last := tx;
	ELSIF NOT q1 AND Tx - last > wait1 THEN
		status := 2;
		q0 := FALSE;
		run := FALSE;
	ELSIF q1 AND tx - last >= delay1 THEN
		step := 2;
		last := tx;
	END_IF;
END_IF;
IF run AND step = 2 THEN
	IF NOT q2 AND in2 AND tx - last <= wait2 THEN
		Q1 := FALSE;
		Q2 := TRUE;
		last := tx;
	ELSIF NOT q2 AND Tx - last > wait2 THEN
		status := 3;
		q1 := FALSE;
		run := FALSE;
	ELSIF q2 AND tx - last >= delay2 THEN
		step := 3;
		last := tx;
	END_IF;
END_IF;
IF run AND step = 3 THEN
	IF NOT q3 AND in3 AND tx - last <= wait3 THEN
		Q2 := FALSE;
		Q3 := TRUE;
		last := tx;
	ELSIF NOT q3 AND Tx - last > wait3 THEN
		status := 4;
		q2 := FALSE;
		run := FALSE;
	ELSIF q3 AND tx - last >= delay3 THEN
		step := 4;
		last := tx;
	END_IF;
END_IF;
IF run AND step = 4 THEN
	IF NOT q4 AND in4 AND tx - last <= wait4 THEN
		Q3 := FALSE;
		Q4 := TRUE;
		last := tx;
	ELSIF NOT q4 AND Tx - last > wait4 THEN
		status := 5;
		q3 := FALSE;
		run := FALSE;
	ELSIF q4 AND tx - last >= delay4 THEN
		step := 5;
		last := tx;
	END_IF;
END_IF;
IF run AND step = 5 THEN
	IF NOT q5 AND in5 AND tx - last <= wait5 THEN
		Q4 := FALSE;
		Q5 := TRUE;
		last := tx;
	ELSIF NOT q5 AND Tx - last > wait5 THEN
		status := 6;
		q4 := FALSE;
		run := FALSE;
	ELSIF q5 AND tx - last >= delay5 THEN
		step := 6;
		last := tx;
	END_IF;
END_IF;
IF run AND step = 6 THEN
	IF NOT q6 AND in6 AND tx - last <= wait6 THEN
		Q5 := FALSE;
		Q6 := TRUE;
		last := tx;
	ELSIF NOT q6 AND Tx - last > wait6 THEN
		status := 7;
		q5 := FALSE;
		run := FALSE;
	ELSIF q6 AND tx - last >= delay6 THEN
		step := 7;
		last := tx;
	END_IF;
END_IF;
IF run AND step = 7 THEN
	IF NOT q7 AND in7 AND tx - last <= wait7 THEN
		Q6 := FALSE;
		Q7 := TRUE;
		last := tx;
	ELSIF NOT q7 AND Tx - last > wait7 THEN
		status := 8;
		q6 := FALSE;
		run := FALSE;
	ELSIF q7 AND tx - last >= delay7 THEN
		step := -1;
		Q7 := FALSE;
		Run := FALSE;
		status := 110;
	END_IF;
END_IF;
QX := q0 OR q1 OR q2 OR q3 OR q4 OR q5 OR q6 OR q7;

(*
hm 1.10.06		rev 1.1
	corrected delay logic to be after event and not before
	added any output

hm 1.12.06		rev 1.2
	corrected failure in sequence logic.
	added init at startup to prevent from initial statuss after start.

hm 17.1.2007		rev 1.3
	changed output fault to status for better compatibility with other modules (ESR)
	added stop on error functionality and setup variable
	default for inputs in0..7 is true.
	renames variable state to step

hm	17.sep 2007	rev 1.4
	replaced time() with T_PLC_MS() for compatibility reasons

hm	13. mar. 2009	rev 1.5
	renamed output any to qx for compatibility resons

*)

END_FUNCTION_BLOCK

// POUs/Logic/generators/TMAX
FUNCTION_BLOCK TMAX
VAR_INPUT
	IN : BOOL;
	PT : TIME;
END_VAR
VAR_OUTPUT
	Q : BOOL;
	Z : BOOL;
END_VAR
VAR
	tx : TIME;
	start : TIME;
	last_in: BOOL;
END_VAR

(*
version 1.0	20. jul. 2008
programmer 	hugo
tested by	oscat

